REGION Network 1
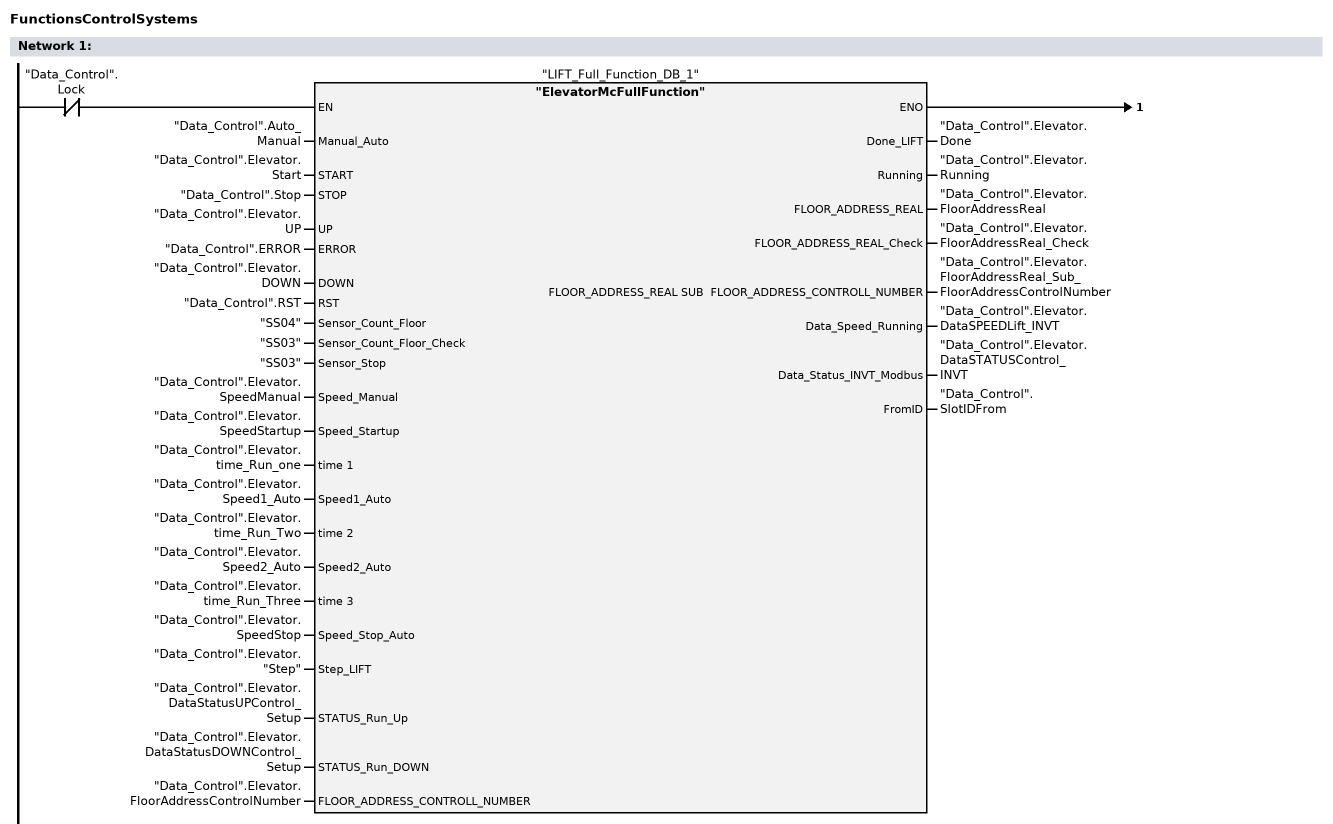
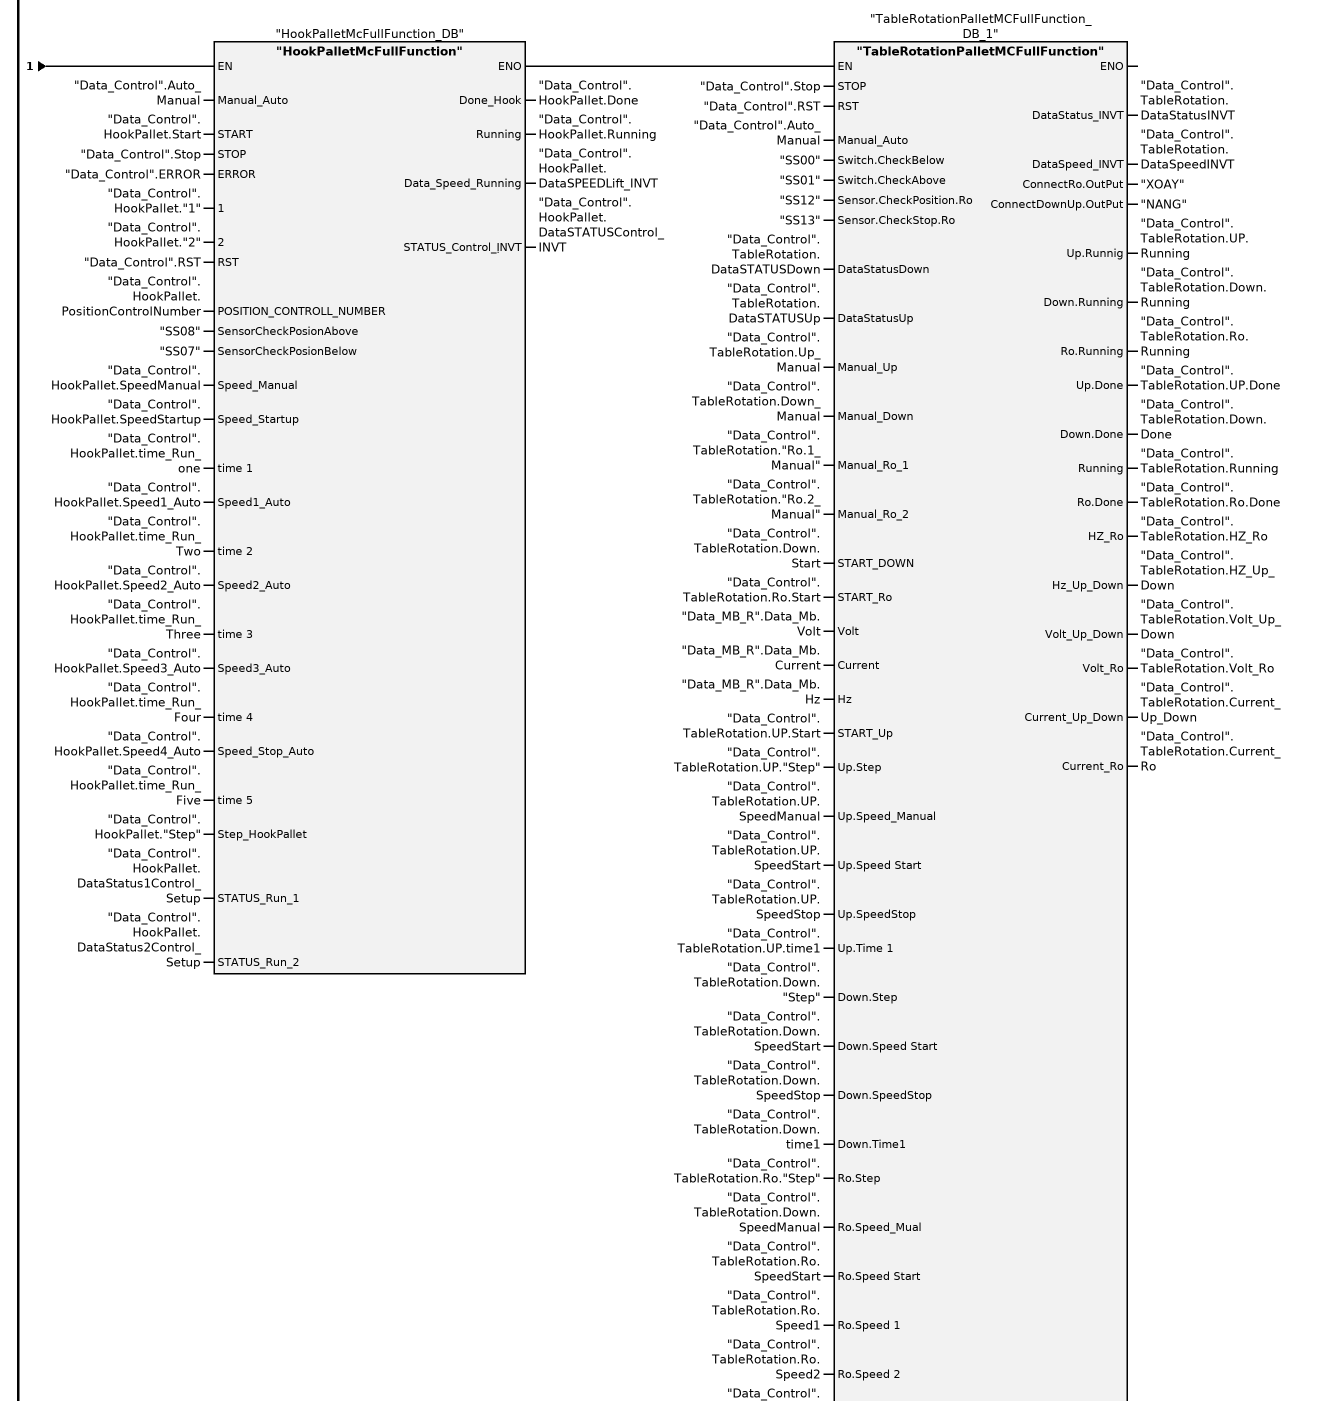
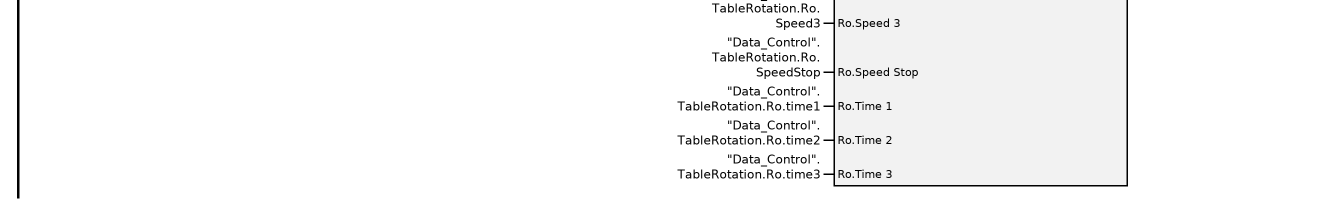
   RUNG wire#powerrail
      I_Contact( "Data_Control".Lock )
      "LIFT_Full_Function_DB_1"(Manual_Auto := "Data_Control".Auto_Manual, START := "Data_Control".Elevator.Start, STOP := "Data_Control".Stop, UP := "Data_Control".Elevator.UP, ERROR := "Data_Control".ERROR, DOWN := "Data_Control".Elevator.DOWN, RST := "Data_Control".RST, Sensor_Count_Floor := "SS04", Sensor_Count_Floor_Check := "SS03", Sensor_Stop := "SS03", Speed_Manual := "Data_Control".Elevator.SpeedManual, Speed_Startup := "Data_Control".Elevator.SpeedStartup, "time 1" := "Data_Control".Elevator.time_Run_one, Speed1_Auto := "Data_Control".Elevator.Speed1_Auto, "time 2" := "Data_Control".Elevator.time_Run_Two, Speed2_Auto := "Data_Control".Elevator.Speed2_Auto, "time 3" := "Data_Control".Elevator.time_Run_Three, Speed_Stop_Auto := "Data_Control".Elevator.SpeedStop, Step_LIFT := "Data_Control".Elevator."Step", STATUS_Run_Up := "Data_Control".Elevator.DataStatusUPControl_Setup, STATUS_Run_DOWN := "Data_Control".Elevator.DataStatusDOWNControl_Setup, FLOOR_ADDRESS_CONTROLL_NUMBER := "Data_Control".Elevator.FloorAddressControlNumber, Done_LIFT => "Data_Control".Elevator.Done, Running => "Data_Control".Elevator.Running, FLOOR_ADDRESS_REAL => "Data_Control".Elevator.FloorAddressReal, FLOOR_ADDRESS_REAL_Check => "Data_Control".Elevator.FloorAddressReal_Check, "FLOOR_ADDRESS_REAL SUB  FLOOR_ADDRESS_CONTROLL_NUMBER" => "Data_Control".Elevator.FloorAddressReal_Sub_FloorAddressControlNumber, Data_Speed_Running => "Data_Control".Elevator.DataSPEEDLift_INVT, Data_Status_INVT_Modbus => "Data_Control".Elevator.DataSTATUSControl_INVT, FromID => "Data_Control".SlotIDFrom)
      "HookPalletMcFullFunction_DB"(Manual_Auto := "Data_Control".Auto_Manual, START := "Data_Control".HookPallet.Start, STOP := "Data_Control".Stop, ERROR := "Data_Control".ERROR, "1" := "Data_Control".HookPallet."1", "2" := "Data_Control".HookPallet."2", RST := "Data_Control".RST, POSITION_CONTROLL_NUMBER := "Data_Control".HookPallet.PositionControlNumber, SensorCheckPosionAbove := "SS08", SensorCheckPosionBelow := "SS07", Speed_Manual := "Data_Control".HookPallet.SpeedManual, Speed_Startup := "Data_Control".HookPallet.SpeedStartup, "time 1" := "Data_Control".HookPallet.time_Run_one, Speed1_Auto := "Data_Control".HookPallet.Speed1_Auto, "time 2" := "Data_Control".HookPallet.time_Run_Two, Speed2_Auto := "Data_Control".HookPallet.Speed2_Auto, "time 3" := "Data_Control".HookPallet.time_Run_Three, Speed3_Auto := "Data_Control".HookPallet.Speed3_Auto, "time 4" := "Data_Control".HookPallet.time_Run_Four, Speed_Stop_Auto := "Data_Control".HookPallet.Speed4_Auto, "time 5" := "Data_Control".HookPallet.time_Run_Five, Step_HookPallet := "Data_Control".HookPallet."Step", STATUS_Run_1 := "Data_Control".HookPallet.DataStatus1Control_Setup, STATUS_Run_2 := "Data_Control".HookPallet.DataStatus2Control_Setup, Done_Hook => "Data_Control".HookPallet.Done, Running => "Data_Control".HookPallet.Running, Data_Speed_Running => "Data_Control".HookPallet.DataSPEEDLift_INVT, STATUS_Control_ỊNVT => "Data_Control".HookPallet.DataSTATUSControl_INVT)
      "TableRotationPalletMCFullFunction_DB_1"(STOP := "Data_Control".Stop, RST := "Data_Control".RST, Manual_Auto := "Data_Control".Auto_Manual, "Switch.CheckBelow" := "SS00", "Switch.CheckAbove" := "SS01", "Sensor.CheckPosition.Ro" := "SS12", "Sensor.CheckStop.Ro" := "SS13", DataStatusDown := "Data_Control".TableRotation.DataSTATUSDown, DataStatusUp := "Data_Control".TableRotation.DataSTATUSUp, Manual_Up := "Data_Control".TableRotation.Up_Manual, Manual_Down := "Data_Control".TableRotation.Down_Manual, Manual_Ro_1 := "Data_Control".TableRotation."Ro.1_Manual", Manual_Ro_2 := "Data_Control".TableRotation."Ro.2_Manual", START_DOWN := "Data_Control".TableRotation.Down.Start, START_Ro := "Data_Control".TableRotation.Ro.Start, Volt := "Data_MB_R".Data_Mb.Volt, Current := "Data_MB_R".Data_Mb.Current, Hz := "Data_MB_R".Data_Mb.Hz, START_Up := "Data_Control".TableRotation.UP.Start, "Up.Step" := "Data_Control".TableRotation.UP."Step", "Up.Speed_Manual" := "Data_Control".TableRotation.UP.SpeedManual, "Up.Speed Start" := "Data_Control".TableRotation.UP.SpeedStart, "Up.SpeedStop" := "Data_Control".TableRotation.UP.SpeedStop, "Up.Time 1" := "Data_Control".TableRotation.UP.time1, "Down.Step" := "Data_Control".TableRotation.Down."Step", "Down.Speed Start" := "Data_Control".TableRotation.Down.SpeedStart, "Down.SpeedStop" := "Data_Control".TableRotation.Down.SpeedStop, "Down.Time1" := "Data_Control".TableRotation.Down.time1, "Ro.Step" := "Data_Control".TableRotation.Ro."Step", "Ro.Speed_Mual" := "Data_Control".TableRotation.Down.SpeedManual, "Ro.Speed Start" := "Data_Control".TableRotation.Ro.SpeedStart, "Ro.Speed 1" := "Data_Control".TableRotation.Ro.Speed1, "Ro.Speed 2" := "Data_Control".TableRotation.Ro.Speed2, "Ro.Speed 3" := "Data_Control".TableRotation.Ro.Speed3, "Ro.Speed Stop" := "Data_Control".TableRotation.Ro.SpeedStop, "Ro.Time 1" := "Data_Control".TableRotation.Ro.time1, "Ro.Time 2" := "Data_Control".TableRotation.Ro.time2, "Ro.Time 3" := "Data_Control".TableRotation.Ro.time3, DataStatus_INVT => "Data_Control".TableRotation.DataStatusINVT, DataSpeed_INVT => "Data_Control".TableRotation.DataSpeedINVT, "ConnectRo.OutPut" => "XOAY", "ConnectDownUp.OutPut" => "NANG", "Up.Runnig" => "Data_Control".TableRotation.UP.Running, "Down.Running" => "Data_Control".TableRotation.Down.Running, "Ro.Running" => "Data_Control".TableRotation.Ro.Running, "Up.Done" => "Data_Control".TableRotation.UP.Done, "Down.Done" => "Data_Control".TableRotation.Down.Done, Running => "Data_Control".TableRotation.Running, "Ro.Done" => "Data_Control".TableRotation.Ro.Done, HZ_Ro => "Data_Control".TableRotation.HZ_Ro, Hz_Up_Down => "Data_Control".TableRotation.HZ_Up_Down, Volt_Up_Down => "Data_Control".TableRotation.Volt_Up_Down, Volt_Ro => "Data_Control".TableRotation.Volt_Ro, Current_Up_Down => "Data_Control".TableRotation.Current_Up_Down, Current_Ro => "Data_Control".TableRotation.Current_Ro)
   END_RUNG
   // the same network as SCL:
   "LIFT_Full_Function_DB_1"(EN := NOT "Data_Control".Lock,   // "ElevatorMcFullFunction"
                           Manual_Auto := "Data_Control".Auto_Manual,
                           START := "Data_Control".Elevator.Start,
                           STOP := "Data_Control".Stop,
                           UP := "Data_Control".Elevator.UP,
                           ERROR := "Data_Control".ERROR,
                           DOWN := "Data_Control".Elevator.DOWN,
                           RST := "Data_Control".RST,
                           Sensor_Count_Floor := "SS04",
                           Sensor_Count_Floor_Check := "SS03",
                           Sensor_Stop := "SS03",
                           Speed_Manual := "Data_Control".Elevator.SpeedManual,
                           Speed_Startup := "Data_Control".Elevator.SpeedStartup,
                           "time 1" := "Data_Control".Elevator.time_Run_one,
                           Speed1_Auto := "Data_Control".Elevator.Speed1_Auto,
                           "time 2" := "Data_Control".Elevator.time_Run_Two,
                           Speed2_Auto := "Data_Control".Elevator.Speed2_Auto,
                           "time 3" := "Data_Control".Elevator.time_Run_Three,
                           Speed_Stop_Auto := "Data_Control".Elevator.SpeedStop,
                           Step_LIFT := "Data_Control".Elevator."Step",
                           STATUS_Run_Up := "Data_Control".Elevator.DataStatusUPControl_Setup,
                           STATUS_Run_DOWN := "Data_Control".Elevator.DataStatusDOWNControl_Setup,
                           FLOOR_ADDRESS_CONTROLL_NUMBER := "Data_Control".Elevator.FloorAddressControlNumber,
                           Done_LIFT => "Data_Control".Elevator.Done,
                           Running => "Data_Control".Elevator.Running,
                           FLOOR_ADDRESS_REAL => "Data_Control".Elevator.FloorAddressReal,
                           FLOOR_ADDRESS_REAL_Check => "Data_Control".Elevator.FloorAddressReal_Check,
                           "FLOOR_ADDRESS_REAL SUB  FLOOR_ADDRESS_CONTROLL_NUMBER" => "Data_Control".Elevator.FloorAddressReal_Sub_FloorAddressControlNumber,
                           Data_Speed_Running => "Data_Control".Elevator.DataSPEEDLift_INVT,
                           Data_Status_INVT_Modbus => "Data_Control".Elevator.DataSTATUSControl_INVT,
                           FromID => "Data_Control".SlotIDFrom,
                           ENO => #_w1);
   "HookPalletMcFullFunction_DB"(EN := #_w1,   // "HookPalletMcFullFunction"
                           Manual_Auto := "Data_Control".Auto_Manual,
                           START := "Data_Control".HookPallet.Start,
                           STOP := "Data_Control".Stop,
                           ERROR := "Data_Control".ERROR,
                           "1" := "Data_Control".HookPallet."1",
                           "2" := "Data_Control".HookPallet."2",
                           RST := "Data_Control".RST,
                           POSITION_CONTROLL_NUMBER := "Data_Control".HookPallet.PositionControlNumber,
                           SensorCheckPosionAbove := "SS08",
                           SensorCheckPosionBelow := "SS07",
                           Speed_Manual := "Data_Control".HookPallet.SpeedManual,
                           Speed_Startup := "Data_Control".HookPallet.SpeedStartup,
                           "time 1" := "Data_Control".HookPallet.time_Run_one,
                           Speed1_Auto := "Data_Control".HookPallet.Speed1_Auto,
                           "time 2" := "Data_Control".HookPallet.time_Run_Two,
                           Speed2_Auto := "Data_Control".HookPallet.Speed2_Auto,
                           "time 3" := "Data_Control".HookPallet.time_Run_Three,
                           Speed3_Auto := "Data_Control".HookPallet.Speed3_Auto,
                           "time 4" := "Data_Control".HookPallet.time_Run_Four,
                           Speed_Stop_Auto := "Data_Control".HookPallet.Speed4_Auto,
                           "time 5" := "Data_Control".HookPallet.time_Run_Five,
                           Step_HookPallet := "Data_Control".HookPallet."Step",
                           STATUS_Run_1 := "Data_Control".HookPallet.DataStatus1Control_Setup,
                           STATUS_Run_2 := "Data_Control".HookPallet.DataStatus2Control_Setup,
                           Done_Hook => "Data_Control".HookPallet.Done,
                           Running => "Data_Control".HookPallet.Running,
                           Data_Speed_Running => "Data_Control".HookPallet.DataSPEEDLift_INVT,
                           STATUS_Control_ỊNVT => "Data_Control".HookPallet.DataSTATUSControl_INVT,
                           ENO => #_w2);
   IF #_w2 THEN
       "TableRotationPalletMCFullFunction_DB_1"(STOP := "Data_Control".Stop,   // "TableRotationPalletMCFullFunction"
                               RST := "Data_Control".RST,
                               Manual_Auto := "Data_Control".Auto_Manual,
                               "Switch.CheckBelow" := "SS00",
                               "Switch.CheckAbove" := "SS01",
                               "Sensor.CheckPosition.Ro" := "SS12",
                               "Sensor.CheckStop.Ro" := "SS13",
                               DataStatusDown := "Data_Control".TableRotation.DataSTATUSDown,
                               DataStatusUp := "Data_Control".TableRotation.DataSTATUSUp,
                               Manual_Up := "Data_Control".TableRotation.Up_Manual,
                               Manual_Down := "Data_Control".TableRotation.Down_Manual,
                               Manual_Ro_1 := "Data_Control".TableRotation."Ro.1_Manual",
                               Manual_Ro_2 := "Data_Control".TableRotation."Ro.2_Manual",
                               START_DOWN := "Data_Control".TableRotation.Down.Start,
                               START_Ro := "Data_Control".TableRotation.Ro.Start,
                               Volt := "Data_MB_R".Data_Mb.Volt,
                               Current := "Data_MB_R".Data_Mb.Current,
                               Hz := "Data_MB_R".Data_Mb.Hz,
                               START_Up := "Data_Control".TableRotation.UP.Start,
                               "Up.Step" := "Data_Control".TableRotation.UP."Step",
                               "Up.Speed_Manual" := "Data_Control".TableRotation.UP.SpeedManual,
                               "Up.Speed Start" := "Data_Control".TableRotation.UP.SpeedStart,
                               "Up.SpeedStop" := "Data_Control".TableRotation.UP.SpeedStop,
                               "Up.Time 1" := "Data_Control".TableRotation.UP.time1,
                               "Down.Step" := "Data_Control".TableRotation.Down."Step",
                               "Down.Speed Start" := "Data_Control".TableRotation.Down.SpeedStart,
                               "Down.SpeedStop" := "Data_Control".TableRotation.Down.SpeedStop,
                               "Down.Time1" := "Data_Control".TableRotation.Down.time1,
                               "Ro.Step" := "Data_Control".TableRotation.Ro."Step",
                               "Ro.Speed_Mual" := "Data_Control".TableRotation.Down.SpeedManual,
                               "Ro.Speed Start" := "Data_Control".TableRotation.Ro.SpeedStart,
                               "Ro.Speed 1" := "Data_Control".TableRotation.Ro.Speed1,
                               "Ro.Speed 2" := "Data_Control".TableRotation.Ro.Speed2,
                               "Ro.Speed 3" := "Data_Control".TableRotation.Ro.Speed3,
                               "Ro.Speed Stop" := "Data_Control".TableRotation.Ro.SpeedStop,
                               "Ro.Time 1" := "Data_Control".TableRotation.Ro.time1,
                               "Ro.Time 2" := "Data_Control".TableRotation.Ro.time2,
                               "Ro.Time 3" := "Data_Control".TableRotation.Ro.time3,
                               DataStatus_INVT => "Data_Control".TableRotation.DataStatusINVT,
                               DataSpeed_INVT => "Data_Control".TableRotation.DataSpeedINVT,
                               "ConnectRo.OutPut" => "XOAY",
                               "ConnectDownUp.OutPut" => "NANG",
                               "Up.Runnig" => "Data_Control".TableRotation.UP.Running,
                               "Down.Running" => "Data_Control".TableRotation.Down.Running,
                               "Ro.Running" => "Data_Control".TableRotation.Ro.Running,
                               "Up.Done" => "Data_Control".TableRotation.UP.Done,
                               "Down.Done" => "Data_Control".TableRotation.Down.Done,
                               Running => "Data_Control".TableRotation.Running,
                               "Ro.Done" => "Data_Control".TableRotation.Ro.Done,
                               HZ_Ro => "Data_Control".TableRotation.HZ_Ro,
                               Hz_Up_Down => "Data_Control".TableRotation.HZ_Up_Down,
                               Volt_Up_Down => "Data_Control".TableRotation.Volt_Up_Down,
                               Volt_Ro => "Data_Control".TableRotation.Volt_Ro,
                               Current_Up_Down => "Data_Control".TableRotation.Current_Up_Down,
                               Current_Ro => "Data_Control".TableRotation.Current_Ro);
   END_IF;
END_REGION
END_FUNCTION_BLOCK

FUNCTION_BLOCK "HookPalletMcFullFunction"   // FB27, LAD
{ S7_Optimized_Access := 'TRUE' }
VERSION : 0.1
   VAR_INPUT
      Manual_Auto : Bool;
      START : Bool;
      STOP : Bool;
      ERROR : Bool;
      "1" : Bool;
      "2" : Bool;
      RST : Bool;
      POSITION_CONTROLL_NUMBER : Int;   // address Elevator use to control
      SensorCheckPosionAbove : Bool;   // it have a Pallet
      SensorCheckPosionBelow : Bool;   // it have not Pallet
      Speed_Manual : Int;
      Speed_Startup : Int;
      "time 1" : Time;
      Speed1_Auto : Int;
      "time 2" : Time;
      Speed2_Auto : Int;
      "time 3" : Time;
      Speed3_Auto : Int;
      "time 4" : Time;
      Speed_Stop_Auto : Int;
      "time 5" : Time;
   END_VAR
   VAR_OUTPUT
      Done_Hook : Bool;
      Running : Bool;   // Lift Running
      Data_Speed_Running : Int;
      STATUS_Control_ỊNVT : Word;
   END_VAR
   VAR_IN_OUT
      Step_HookPallet : Int;   // steps used to control
      STATUS_Run_1 : Word := 16#0002;   // Set_Up Run R/F
      STATUS_Run_2 : Word := 16#0004;   // Set_Up Run R/F
   END_VAR
   VAR_TEMP   // added for the SCL form of the ladder/FBD networks
      _w1 : Bool;
   END_VAR
BEGIN

REGION Network 1
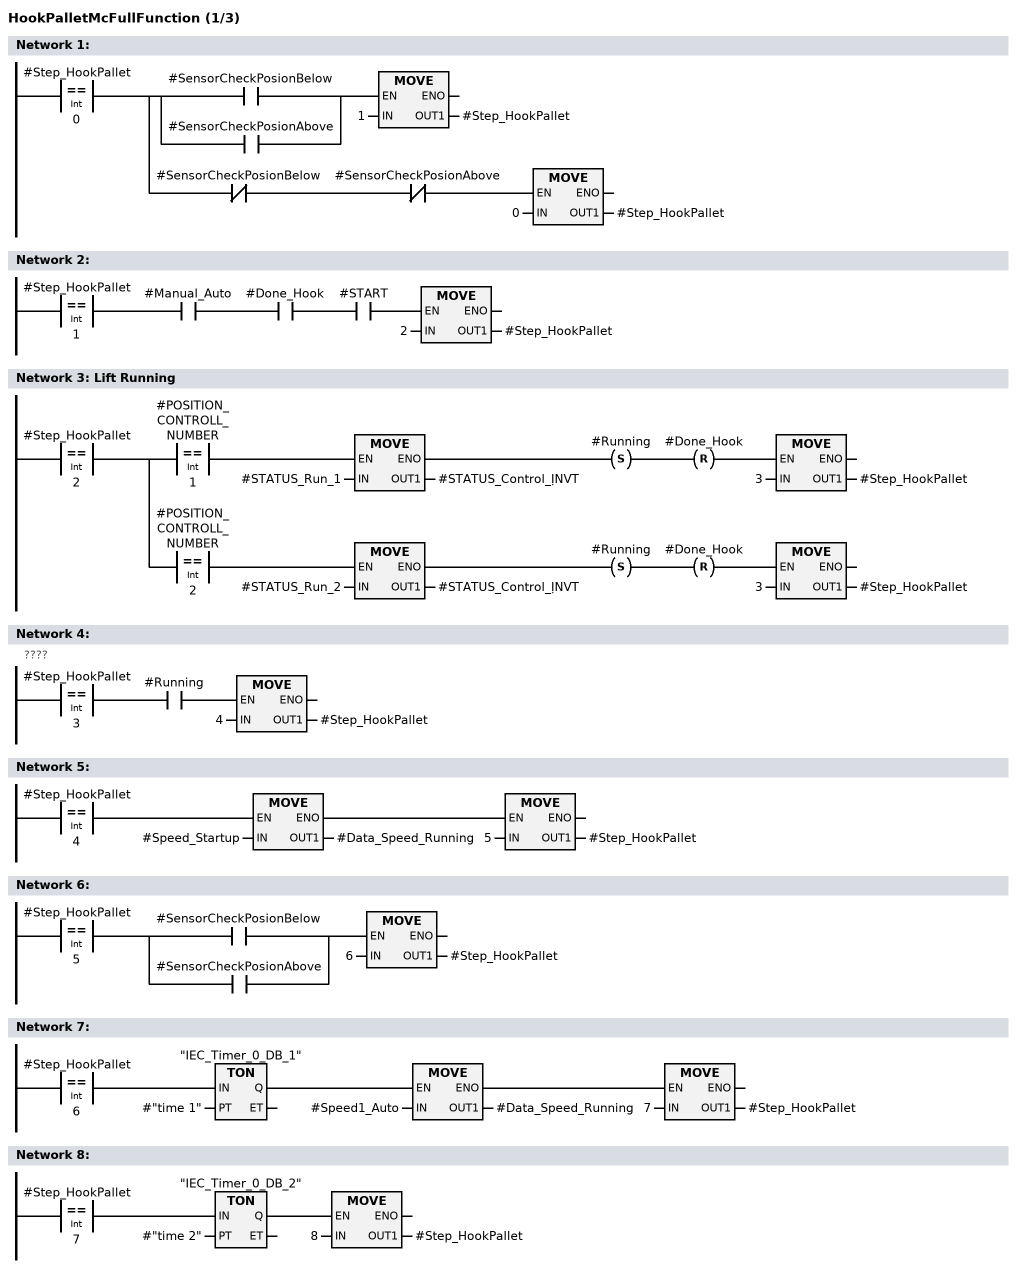
   RUNG wire#powerrail
      { S7_Templates := "SrcType := Int" } EQ_Contact(in1 := #Step_HookPallet, in2 := 0)
      wire#w1
      Contact( #SensorCheckPosionBelow )
      wire#w2
      Move(in := 1, out1 => #Step_HookPallet)
   END_RUNG
   RUNG wire#w1
      Contact( #SensorCheckPosionAbove )
   END_RUNG wire#w2
   RUNG wire#w1
      I_Contact( #SensorCheckPosionBelow )
      I_Contact( #SensorCheckPosionAbove )
      Move(in := 0, out1 => #Step_HookPallet)
   END_RUNG
   // the same network as SCL:
   #_w1 := #Step_HookPallet = 0;
   IF #_w1 AND (#SensorCheckPosionBelow OR #SensorCheckPosionAbove) THEN #Step_HookPallet := 1; END_IF;
   IF #_w1 AND NOT #SensorCheckPosionBelow AND NOT #SensorCheckPosionAbove THEN
       #Step_HookPallet := 0;
   END_IF;
END_REGION

REGION Network 2
   RUNG wire#powerrail
      { S7_Templates := "SrcType := Int" } EQ_Contact(in1 := #Step_HookPallet, in2 := 1)
      Contact( #Manual_Auto )
      Contact( #Done_Hook )
      Contact( #START )
      Move(in := 2, out1 => #Step_HookPallet)
   END_RUNG
   // the same network as SCL:
   IF (#Step_HookPallet = 1) AND #Manual_Auto AND #Done_Hook AND #START THEN #Step_HookPallet := 2; END_IF;
END_REGION

REGION Network 3: Lift Running
   RUNG wire#powerrail
      { S7_Templates := "SrcType := Int" } EQ_Contact(in1 := #Step_HookPallet, in2 := 2)
      wire#w1
      { S7_Templates := "SrcType := Int" } EQ_Contact(in1 := #POSITION_CONTROLL_NUMBER, in2 := 1)
      Move(in := #STATUS_Run_1, out1 => #STATUS_Control_ỊNVT)
      S_Coil( #Running )
      R_Coil( #Done_Hook )
      Move(in := 3, out1 => #Step_HookPallet)
   END_RUNG
   RUNG wire#w1
      { S7_Templates := "SrcType := Int" } EQ_Contact(in1 := #POSITION_CONTROLL_NUMBER, in2 := 2)
      Move(in := #STATUS_Run_2, out1 => #STATUS_Control_ỊNVT)
      S_Coil( #Running )
      R_Coil( #Done_Hook )
      Move(in := 3, out1 => #Step_HookPallet)
   END_RUNG
   // the same network as SCL:
   #_w1 := #Step_HookPallet = 2;
   IF #_w1 AND (#POSITION_CONTROLL_NUMBER = 1) THEN
       #STATUS_Control_ỊNVT := #STATUS_Run_1;
       #Running := TRUE;
       #Done_Hook := FALSE;
       #Step_HookPallet := 3;
   END_IF;
   IF #_w1 AND (#POSITION_CONTROLL_NUMBER = 2) THEN
       #STATUS_Control_ỊNVT := #STATUS_Run_2;
       #Running := TRUE;
       #Done_Hook := FALSE;
       #Step_HookPallet := 3;
   END_IF;
END_REGION

REGION Network 4
   // ????
   RUNG wire#powerrail
      { S7_Templates := "SrcType := Int" } EQ_Contact(in1 := #Step_HookPallet, in2 := 3)
      Contact( #Running )
      Move(in := 4, out1 => #Step_HookPallet)
   END_RUNG
   // the same network as SCL:
   IF (#Step_HookPallet = 3) AND #Running THEN #Step_HookPallet := 4; END_IF;
END_REGION

REGION Network 5
   RUNG wire#powerrail
      { S7_Templates := "SrcType := Int" } EQ_Contact(in1 := #Step_HookPallet, in2 := 4)
      Move(in := #Speed_Startup, out1 => #Data_Speed_Running)
      Move(in := 5, out1 => #Step_HookPallet)
   END_RUNG
   // the same network as SCL:
   IF #Step_HookPallet = 4 THEN
       #Data_Speed_Running := #Speed_Startup;
       #Step_HookPallet := 5;
   END_IF;
END_REGION

REGION Network 6
   RUNG wire#powerrail
      { S7_Templates := "SrcType := Int" } EQ_Contact(in1 := #Step_HookPallet, in2 := 5)
      wire#w1
      Contact( #SensorCheckPosionBelow )
      wire#w2
      Move(in := 6, out1 => #Step_HookPallet)
   END_RUNG
   RUNG wire#w1
      Contact( #SensorCheckPosionAbove )
   END_RUNG wire#w2
   // the same network as SCL:
   IF (#Step_HookPallet = 5) AND (#SensorCheckPosionBelow OR #SensorCheckPosionAbove) THEN
       #Step_HookPallet := 6;
   END_IF;
END_REGION

REGION Network 7
   "IEC_Timer_0_DB_1".TON(IN := #Step_HookPallet = 6, PT := #"time 1");
   IF "IEC_Timer_0_DB_1".Q THEN
       #Data_Speed_Running := #Speed1_Auto;
       #Step_HookPallet := 7;
   END_IF;
END_REGION

REGION Network 8
   "IEC_Timer_0_DB_2".TON(IN := #Step_HookPallet = 7, PT := #"time 2");
   IF "IEC_Timer_0_DB_2".Q THEN #Step_HookPallet := 8; END_IF;
END_REGION

REGION Network 9
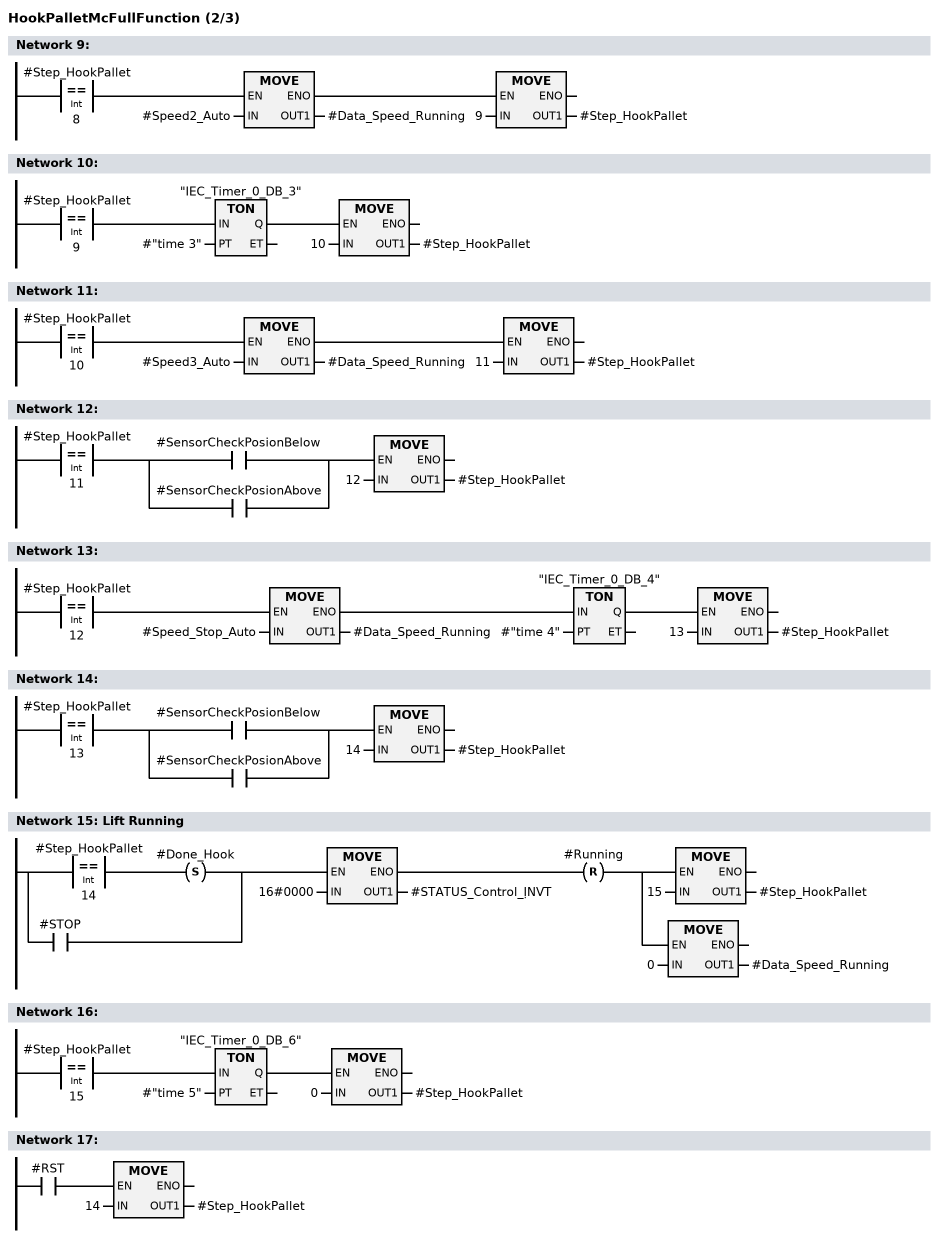
   RUNG wire#powerrail
      { S7_Templates := "SrcType := Int" } EQ_Contact(in1 := #Step_HookPallet, in2 := 8)
      Move(in := #Speed2_Auto, out1 => #Data_Speed_Running)
      Move(in := 9, out1 => #Step_HookPallet)
   END_RUNG
   // the same network as SCL:
   IF #Step_HookPallet = 8 THEN
       #Data_Speed_Running := #Speed2_Auto;
       #Step_HookPallet := 9;
   END_IF;
END_REGION

REGION Network 10
   "IEC_Timer_0_DB_3".TON(IN := #Step_HookPallet = 9, PT := #"time 3");
   IF "IEC_Timer_0_DB_3".Q THEN #Step_HookPallet := 10; END_IF;
END_REGION

REGION Network 11
   RUNG wire#powerrail
      { S7_Templates := "SrcType := Int" } EQ_Contact(in1 := #Step_HookPallet, in2 := 10)
      Move(in := #Speed3_Auto, out1 => #Data_Speed_Running)
      Move(in := 11, out1 => #Step_HookPallet)
   END_RUNG
   // the same network as SCL:
   IF #Step_HookPallet = 10 THEN
       #Data_Speed_Running := #Speed3_Auto;
       #Step_HookPallet := 11;
   END_IF;
END_REGION

REGION Network 12
   RUNG wire#powerrail
      { S7_Templates := "SrcType := Int" } EQ_Contact(in1 := #Step_HookPallet, in2 := 11)
      wire#w1
      Contact( #SensorCheckPosionBelow )
      wire#w2
      Move(in := 12, out1 => #Step_HookPallet)
   END_RUNG
   RUNG wire#w1
      Contact( #SensorCheckPosionAbove )
   END_RUNG wire#w2
   // the same network as SCL:
   IF (#Step_HookPallet = 11) AND (#SensorCheckPosionBelow OR #SensorCheckPosionAbove) THEN
       #Step_HookPallet := 12;
   END_IF;
END_REGION

REGION Network 13
   #_w1 := #Step_HookPallet = 12;
   IF #_w1 THEN #Data_Speed_Running := #Speed_Stop_Auto; END_IF;
   "IEC_Timer_0_DB_4".TON(IN := #_w1, PT := #"time 4");
   IF "IEC_Timer_0_DB_4".Q THEN #Step_HookPallet := 13; END_IF;
END_REGION

REGION Network 14
   RUNG wire#powerrail
      { S7_Templates := "SrcType := Int" } EQ_Contact(in1 := #Step_HookPallet, in2 := 13)
      wire#w1
      Contact( #SensorCheckPosionBelow )
      wire#w2
      Move(in := 14, out1 => #Step_HookPallet)
   END_RUNG
   RUNG wire#w1
      Contact( #SensorCheckPosionAbove )
   END_RUNG wire#w2
   // the same network as SCL:
   IF (#Step_HookPallet = 13) AND (#SensorCheckPosionBelow OR #SensorCheckPosionAbove) THEN
       #Step_HookPallet := 14;
   END_IF;
END_REGION

REGION Network 15: Lift Running
   RUNG wire#powerrail
      { S7_Templates := "SrcType := Int" } EQ_Contact(in1 := #Step_HookPallet, in2 := 14)
      S_Coil( #Done_Hook )
      wire#w1
      Move(in := 16#0000, out1 => #STATUS_Control_ỊNVT)
      R_Coil( #Running )
      wire#w2
      Move(in := 15, out1 => #Step_HookPallet)
   END_RUNG
   RUNG wire#powerrail
      Contact( #STOP )
   END_RUNG wire#w1
   RUNG wire#w2
      Move(in := 0, out1 => #Data_Speed_Running)
   END_RUNG
   // the same network as SCL:
   #_w1 := #Step_HookPallet = 14;
   IF #_w1 THEN #Done_Hook := TRUE; END_IF;
   IF #_w1 OR #STOP THEN
       #STATUS_Control_ỊNVT := 16#0000;
       #Running := FALSE;
       #Step_HookPallet := 15;
       #Data_Speed_Running := 0;
   END_IF;
END_REGION

REGION Network 16
   "IEC_Timer_0_DB_6".TON(IN := #Step_HookPallet = 15, PT := #"time 5");
   IF "IEC_Timer_0_DB_6".Q THEN #Step_HookPallet := 0; END_IF;
END_REGION

REGION Network 17
   RUNG wire#powerrail
      Contact( #RST )
      Move(in := 14, out1 => #Step_HookPallet)
   END_RUNG
   // the same network as SCL:
   IF #RST THEN #Step_HookPallet := 14; END_IF;
END_REGION

REGION Network 18
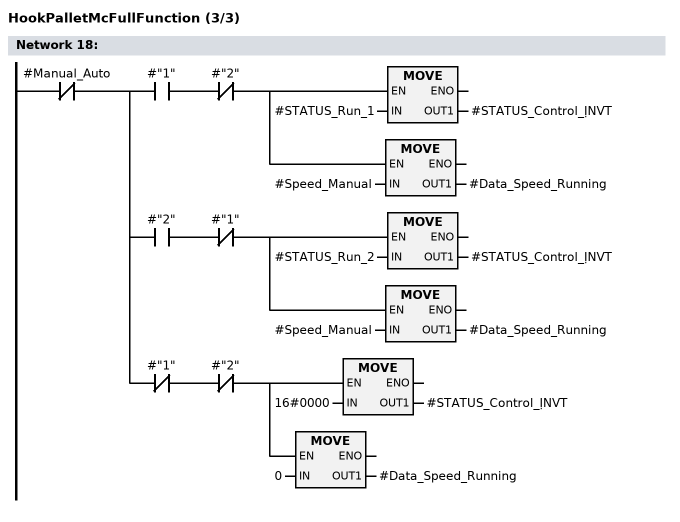
   RUNG wire#powerrail
      I_Contact( #Manual_Auto )
      wire#w1
      Contact( #"1" )
      I_Contact( #"2" )
      wire#w2
      Move(in := #STATUS_Run_1, out1 => #STATUS_Control_ỊNVT)
   END_RUNG
   RUNG wire#w2
      Move(in := #Speed_Manual, out1 => #Data_Speed_Running)
   END_RUNG
   RUNG wire#w1
      Contact( #"2" )
      I_Contact( #"1" )
      wire#w3
      Move(in := #STATUS_Run_2, out1 => #STATUS_Control_ỊNVT)
   END_RUNG
   RUNG wire#w3
      Move(in := #Speed_Manual, out1 => #Data_Speed_Running)
   END_RUNG
   RUNG wire#w1
      I_Contact( #"1" )
      I_Contact( #"2" )
      wire#w4
      Move(in := 16#0000, out1 => #STATUS_Control_ỊNVT)
   END_RUNG
   RUNG wire#w4
      Move(in := 0, out1 => #Data_Speed_Running)
   END_RUNG
   // the same network as SCL:
   IF NOT #Manual_Auto AND #"1" AND NOT #"2" THEN
       #STATUS_Control_ỊNVT := #STATUS_Run_1;
       #Data_Speed_Running := #Speed_Manual;
   END_IF;
   IF NOT #Manual_Auto AND #"2" AND NOT #"1" THEN
       #STATUS_Control_ỊNVT := #STATUS_Run_2;
       #Data_Speed_Running := #Speed_Manual;
   END_IF;
   IF NOT #Manual_Auto AND NOT #"1" AND NOT #"2" THEN
       #STATUS_Control_ỊNVT := 16#0000;
       #Data_Speed_Running := 0;
   END_IF;
END_REGION
END_FUNCTION_BLOCK

FUNCTION_BLOCK "TableRotationPalletMCFullFunction"   // FB28, LAD
{ S7_Optimized_Access := 'TRUE' }
VERSION : 0.1
   VAR_INPUT
      STOP : Bool;
      RST : Bool;
      Manual_Auto : Bool;
      "Switch.CheckBelow" : Bool;
      "Switch.CheckAbove" : Bool;
      "Sensor.CheckPosition.Ro" : Bool;
      "Sensor.CheckStop.Ro" : Bool;
      DataStatusDown : Word := 16#0002;
      DataStatusUp : Word := 16#0004;
      Manual_Up : Bool;
      Manual_Down : Bool;
      Manual_Ro_1 : Bool;
      Manual_Ro_2 : Bool;
      START_DOWN : Bool;
      START_Ro : Bool;
      Volt : Int;
      Current : Int;
      Hz : Int;
      START_Up : Bool;
   END_VAR
   VAR_OUTPUT
      DataStatus_INVT : Word;
      DataSpeed_INVT : Int;
      "ConnectRo.OutPut" : Bool;
      "ConnectDownUp.OutPut" : Bool;
      "Up.Runnig" : Bool;
      "Down.Running" : Bool;
      "Ro.Running" : Bool;
      "Up.Done" : Bool;
      "Down.Done" : Bool;
      Running : Bool;
      "Ro.Done" : Bool;
      HZ_Ro : Int;
      Hz_Up_Down : Int;
      Volt_Up_Down : Int;
      Volt_Ro : Int;
      Current_Up_Down : Int;
      Current_Ro : Int;
   END_VAR
   VAR_IN_OUT
      "Up.Step" : Int;
      "Up.Speed_Manual" : Int;
      "Up.Speed Start" : Int;
      "Up.SpeedStop" : Int;
      "Up.Time 1" : Time;
      "Down.Step" : Int;
      "Down.Speed Start" : Int;
      "Down.SpeedStop" : Int;
      "Down.Time1" : Time;
      "Ro.Step" : Int;
      "Ro.Speed_Mual" : Int;
      "Ro.Speed Start" : Int;
      "Ro.Speed 1" : Int;
      "Ro.Speed 2" : Int;
      "Ro.Speed 3" : Int;
      "Ro.Speed Stop" : Int;
      "Ro.Time 1" : Time;
      "Ro.Time 2" : Time;
      "Ro.Time 3" : Time;
   END_VAR
   VAR_TEMP   // added for the SCL form of the ladder/FBD networks
      _w1 : Bool;
      _w2 : Bool;
   END_VAR
BEGIN

REGION Network 1
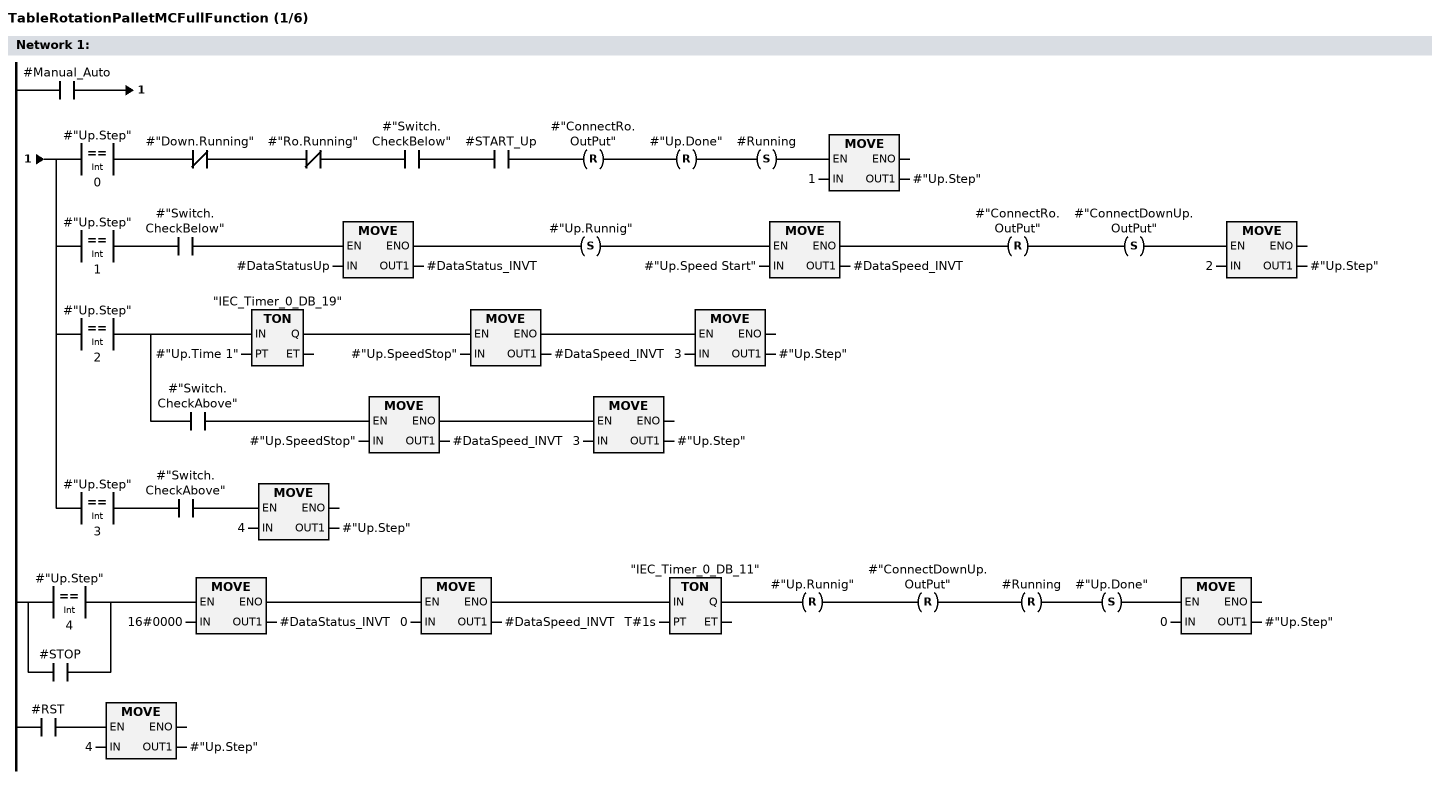
   IF #Manual_Auto AND (#"Up.Step" = 0) AND NOT #"Down.Running" AND NOT #"Ro.Running" AND #"Switch.CheckBelow" AND #START_Up THEN
       #"ConnectRo.OutPut" := FALSE;
       #"Up.Done" := FALSE;
       #Running := TRUE;
       #"Up.Step" := 1;
   END_IF;
   IF #Manual_Auto AND (#"Up.Step" = 1) AND #"Switch.CheckBelow" THEN
       #DataStatus_INVT := #DataStatusUp;
       #"Up.Runnig" := TRUE;
       #DataSpeed_INVT := #"Up.Speed Start";
       #"ConnectRo.OutPut" := FALSE;
       #"ConnectDownUp.OutPut" := TRUE;
       #"Up.Step" := 2;
   END_IF;
   #_w1 := #Manual_Auto AND (#"Up.Step" = 2);
   "IEC_Timer_0_DB_19".TON(IN := #_w1, PT := #"Up.Time 1");
   IF "IEC_Timer_0_DB_19".Q THEN
       #DataSpeed_INVT := #"Up.SpeedStop";
       #"Up.Step" := 3;
   END_IF;
   IF #_w1 AND #"Switch.CheckAbove" THEN
       #DataSpeed_INVT := #"Up.SpeedStop";
       #"Up.Step" := 3;
   END_IF;
   IF #Manual_Auto AND (#"Up.Step" = 3) AND #"Switch.CheckAbove" THEN #"Up.Step" := 4; END_IF;
   #_w2 := (#"Up.Step" = 4) OR #STOP;
   IF #_w2 THEN
       #DataStatus_INVT := 16#0000;
       #DataSpeed_INVT := 0;
   END_IF;
   "IEC_Timer_0_DB_11".TON(IN := #_w2, PT := T#1s);
   IF "IEC_Timer_0_DB_11".Q THEN
       #"Up.Runnig" := FALSE;
       #"ConnectDownUp.OutPut" := FALSE;
       #Running := FALSE;
       #"Up.Done" := TRUE;
       #"Up.Step" := 0;
   END_IF;
   IF #RST THEN #"Up.Step" := 4; END_IF;
END_REGION

REGION Network 2
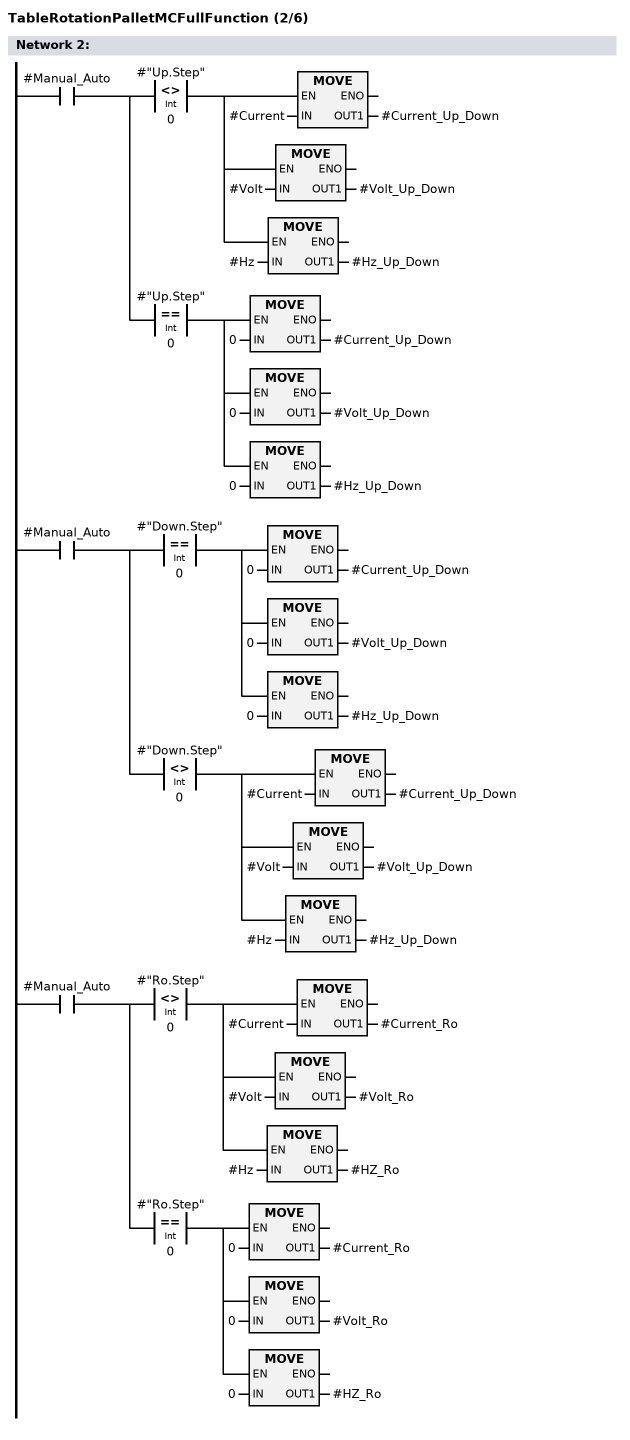
   RUNG wire#powerrail
      Contact( #Manual_Auto )
      wire#w1
      { S7_Templates := "SrcType := Int" } NE_Contact(in1 := #"Up.Step", in2 := 0)
      wire#w2
      Move(in := #Current, out1 => #Current_Up_Down)
   END_RUNG
   RUNG wire#w2
      Move(in := #Volt, out1 => #Volt_Up_Down)
   END_RUNG
   RUNG wire#w2
      Move(in := #Hz, out1 => #Hz_Up_Down)
   END_RUNG
   RUNG wire#w1
      { S7_Templates := "SrcType := Int" } EQ_Contact(in1 := #"Up.Step", in2 := 0)
      wire#w3
      Move(in := 0, out1 => #Current_Up_Down)
   END_RUNG
   RUNG wire#w3
      Move(in := 0, out1 => #Volt_Up_Down)
   END_RUNG
   RUNG wire#w3
      Move(in := 0, out1 => #Hz_Up_Down)
   END_RUNG
   RUNG wire#powerrail
      Contact( #Manual_Auto )
      wire#w4
      { S7_Templates := "SrcType := Int" } EQ_Contact(in1 := #"Down.Step", in2 := 0)
      wire#w5
      Move(in := 0, out1 => #Current_Up_Down)
   END_RUNG
   RUNG wire#w5
      Move(in := 0, out1 => #Volt_Up_Down)
   END_RUNG
   RUNG wire#w5
      Move(in := 0, out1 => #Hz_Up_Down)
   END_RUNG
   RUNG wire#w4
      { S7_Templates := "SrcType := Int" } NE_Contact(in1 := #"Down.Step", in2 := 0)
      wire#w6
      Move(in := #Current, out1 => #Current_Up_Down)
   END_RUNG
   RUNG wire#w6
      Move(in := #Volt, out1 => #Volt_Up_Down)
   END_RUNG
   RUNG wire#w6
      Move(in := #Hz, out1 => #Hz_Up_Down)
   END_RUNG
   RUNG wire#powerrail
      Contact( #Manual_Auto )
      wire#w7
      { S7_Templates := "SrcType := Int" } NE_Contact(in1 := #"Ro.Step", in2 := 0)
      wire#w8
      Move(in := #Current, out1 => #Current_Ro)
   END_RUNG
   RUNG wire#w8
      Move(in := #Volt, out1 => #Volt_Ro)
   END_RUNG
   RUNG wire#w8
      Move(in := #Hz, out1 => #HZ_Ro)
   END_RUNG
   RUNG wire#w7
      { S7_Templates := "SrcType := Int" } EQ_Contact(in1 := #"Ro.Step", in2 := 0)
      wire#w9
      Move(in := 0, out1 => #Current_Ro)
   END_RUNG
   RUNG wire#w9
      Move(in := 0, out1 => #Volt_Ro)
   END_RUNG
   RUNG wire#w9
      Move(in := 0, out1 => #HZ_Ro)
   END_RUNG
   // the same network as SCL:
   IF #Manual_Auto AND (#"Up.Step" <> 0) THEN
       #Current_Up_Down := #Current;
       #Volt_Up_Down := #Volt;
       #Hz_Up_Down := #Hz;
   END_IF;
   IF #Manual_Auto AND (#"Up.Step" = 0) THEN
       #Current_Up_Down := 0;
       #Volt_Up_Down := 0;
       #Hz_Up_Down := 0;
   END_IF;
   IF #Manual_Auto AND (#"Down.Step" = 0) THEN
       #Current_Up_Down := 0;
       #Volt_Up_Down := 0;
       #Hz_Up_Down := 0;
   END_IF;
   IF #Manual_Auto AND (#"Down.Step" <> 0) THEN
       #Current_Up_Down := #Current;
       #Volt_Up_Down := #Volt;
       #Hz_Up_Down := #Hz;
   END_IF;
   IF #Manual_Auto AND (#"Ro.Step" <> 0) THEN
       #Current_Ro := #Current;
       #Volt_Ro := #Volt;
       #HZ_Ro := #Hz;
   END_IF;
   IF #Manual_Auto AND (#"Ro.Step" = 0) THEN
       #Current_Ro := 0;
       #Volt_Ro := 0;
       #HZ_Ro := 0;
   END_IF;
END_REGION

REGION Network 3
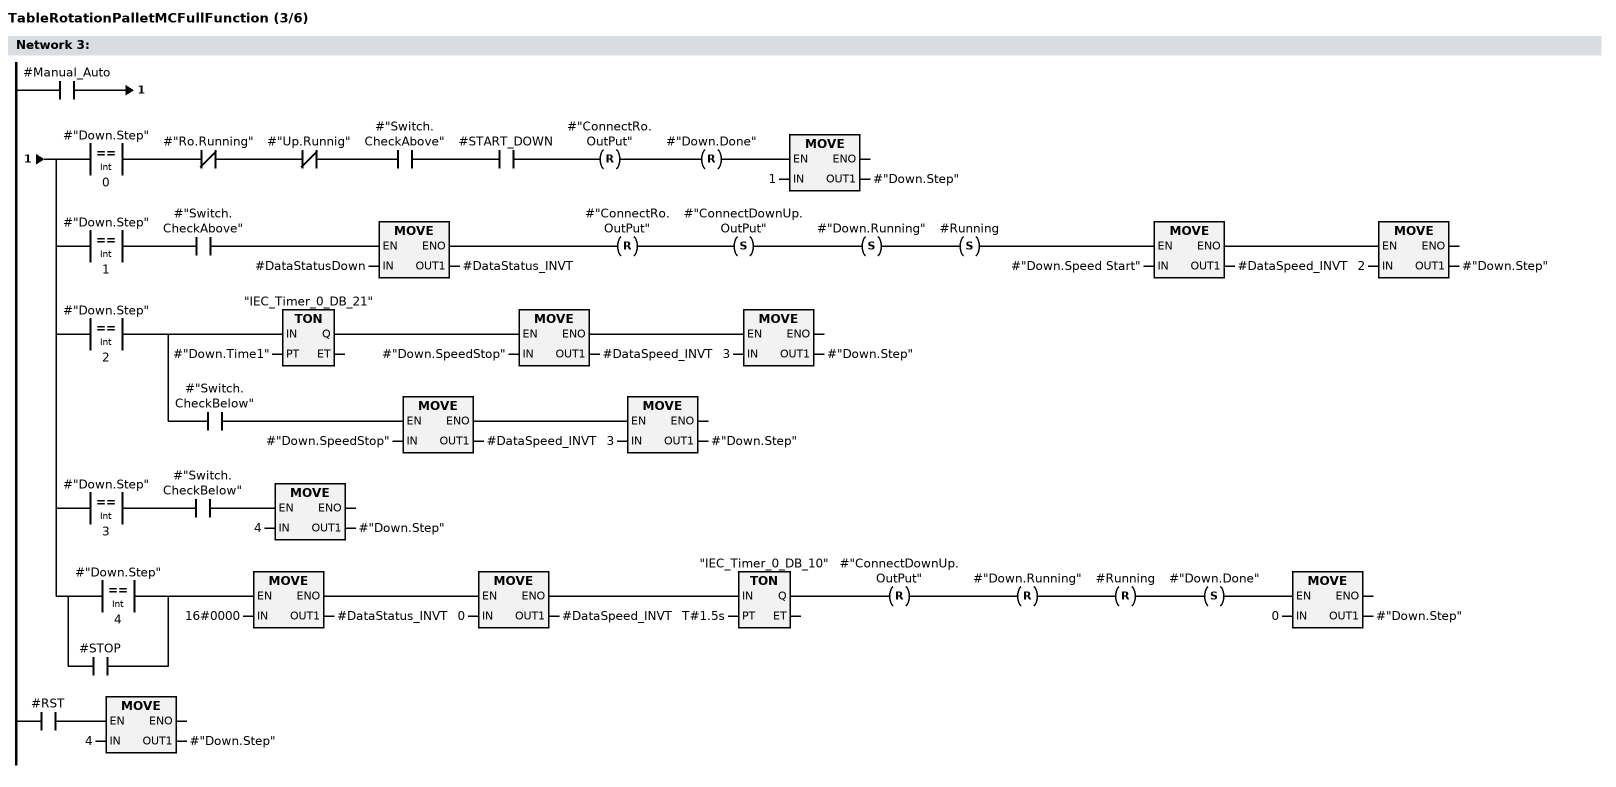
   IF #Manual_Auto AND (#"Down.Step" = 0) AND NOT #"Ro.Running" AND NOT #"Up.Runnig" AND #"Switch.CheckAbove" AND #START_DOWN THEN
       #"ConnectRo.OutPut" := FALSE;
       #"Down.Done" := FALSE;
       #"Down.Step" := 1;
   END_IF;
   IF #Manual_Auto AND (#"Down.Step" = 1) AND #"Switch.CheckAbove" THEN
       #DataStatus_INVT := #DataStatusDown;
       #"ConnectRo.OutPut" := FALSE;
       #"ConnectDownUp.OutPut" := TRUE;
       #"Down.Running" := TRUE;
       #Running := TRUE;
       #DataSpeed_INVT := #"Down.Speed Start";
       #"Down.Step" := 2;
   END_IF;
   #_w1 := #Manual_Auto AND (#"Down.Step" = 2);
   "IEC_Timer_0_DB_21".TON(IN := #_w1, PT := #"Down.Time1");
   IF "IEC_Timer_0_DB_21".Q THEN
       #DataSpeed_INVT := #"Down.SpeedStop";
       #"Down.Step" := 3;
   END_IF;
   IF #_w1 AND #"Switch.CheckBelow" THEN
       #DataSpeed_INVT := #"Down.SpeedStop";
       #"Down.Step" := 3;
   END_IF;
   IF #Manual_Auto AND (#"Down.Step" = 3) AND #"Switch.CheckBelow" THEN #"Down.Step" := 4; END_IF;
   #_w2 := #Manual_Auto AND ((#"Down.Step" = 4) OR #STOP);
   IF #_w2 THEN
       #DataStatus_INVT := 16#0000;
       #DataSpeed_INVT := 0;
   END_IF;
   "IEC_Timer_0_DB_10".TON(IN := #_w2, PT := T#1.5s);
   IF "IEC_Timer_0_DB_10".Q THEN
       #"ConnectDownUp.OutPut" := FALSE;
       #"Down.Running" := FALSE;
       #Running := FALSE;
       #"Down.Done" := TRUE;
       #"Down.Step" := 0;
   END_IF;
   IF #RST THEN #"Down.Step" := 4; END_IF;
END_REGION

REGION Network 5
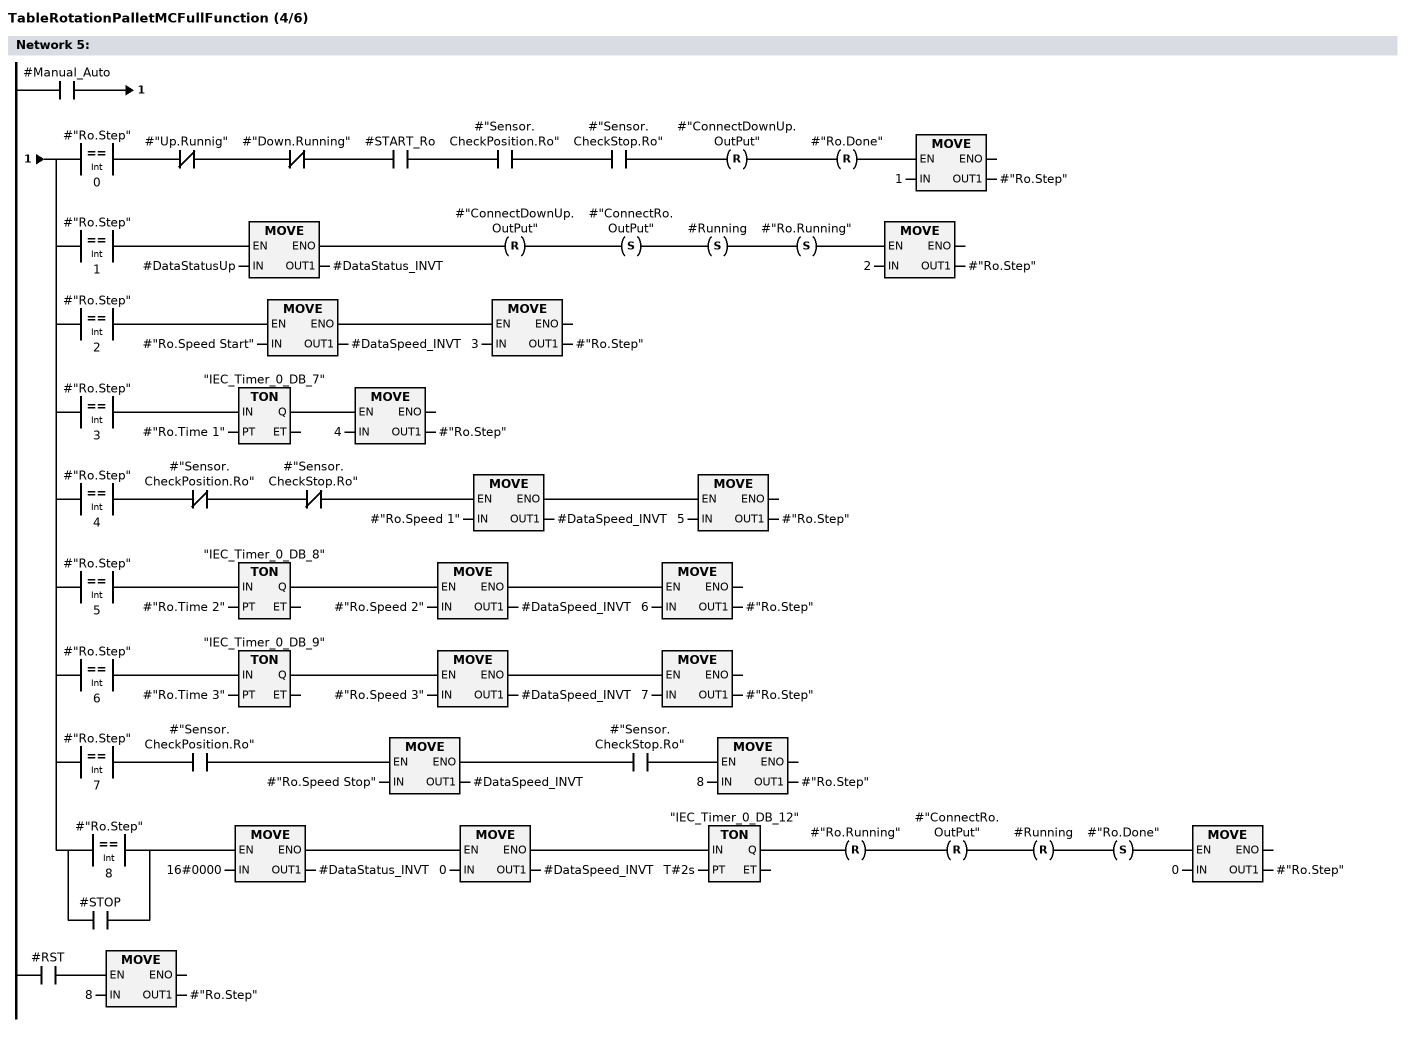
   IF #Manual_Auto AND (#"Ro.Step" = 0) AND NOT #"Up.Runnig" AND NOT #"Down.Running" AND #START_Ro AND #"Sensor.CheckPosition.Ro" AND #"Sensor.CheckStop.Ro" THEN
       #"ConnectDownUp.OutPut" := FALSE;
       #"Ro.Done" := FALSE;
       #"Ro.Step" := 1;
   END_IF;
   IF #Manual_Auto AND (#"Ro.Step" = 1) THEN
       #DataStatus_INVT := #DataStatusUp;
       #"ConnectDownUp.OutPut" := FALSE;
       #"ConnectRo.OutPut" := TRUE;
       #Running := TRUE;
       #"Ro.Running" := TRUE;
       #"Ro.Step" := 2;
   END_IF;
   IF #Manual_Auto AND (#"Ro.Step" = 2) THEN
       #DataSpeed_INVT := #"Ro.Speed Start";
       #"Ro.Step" := 3;
   END_IF;
   "IEC_Timer_0_DB_7".TON(IN := #Manual_Auto AND (#"Ro.Step" = 3), PT := #"Ro.Time 1");
   IF "IEC_Timer_0_DB_7".Q THEN #"Ro.Step" := 4; END_IF;
   IF #Manual_Auto AND (#"Ro.Step" = 4) AND NOT #"Sensor.CheckPosition.Ro" AND NOT #"Sensor.CheckStop.Ro" THEN
       #DataSpeed_INVT := #"Ro.Speed 1";
       #"Ro.Step" := 5;
   END_IF;
   "IEC_Timer_0_DB_8".TON(IN := #Manual_Auto AND (#"Ro.Step" = 5), PT := #"Ro.Time 2");
   IF "IEC_Timer_0_DB_8".Q THEN
       #DataSpeed_INVT := #"Ro.Speed 2";
       #"Ro.Step" := 6;
   END_IF;
   "IEC_Timer_0_DB_9".TON(IN := #Manual_Auto AND (#"Ro.Step" = 6), PT := #"Ro.Time 3");
   IF "IEC_Timer_0_DB_9".Q THEN
       #DataSpeed_INVT := #"Ro.Speed 3";
       #"Ro.Step" := 7;
   END_IF;
   #_w1 := #Manual_Auto AND (#"Ro.Step" = 7) AND #"Sensor.CheckPosition.Ro";
   IF #_w1 THEN #DataSpeed_INVT := #"Ro.Speed Stop"; END_IF;
   IF #_w1 AND #"Sensor.CheckStop.Ro" THEN #"Ro.Step" := 8; END_IF;
   #_w2 := #Manual_Auto AND ((#"Ro.Step" = 8) OR #STOP);
   IF #_w2 THEN
       #DataStatus_INVT := 16#0000;
       #DataSpeed_INVT := 0;
   END_IF;
   "IEC_Timer_0_DB_12".TON(IN := #_w2, PT := T#2s);
   IF "IEC_Timer_0_DB_12".Q THEN
       #"Ro.Running" := FALSE;
       #"ConnectRo.OutPut" := FALSE;
       #Running := FALSE;
       #"Ro.Done" := TRUE;
       #"Ro.Step" := 0;
   END_IF;
   IF #RST THEN #"Ro.Step" := 8; END_IF;
END_REGION

REGION Network 8
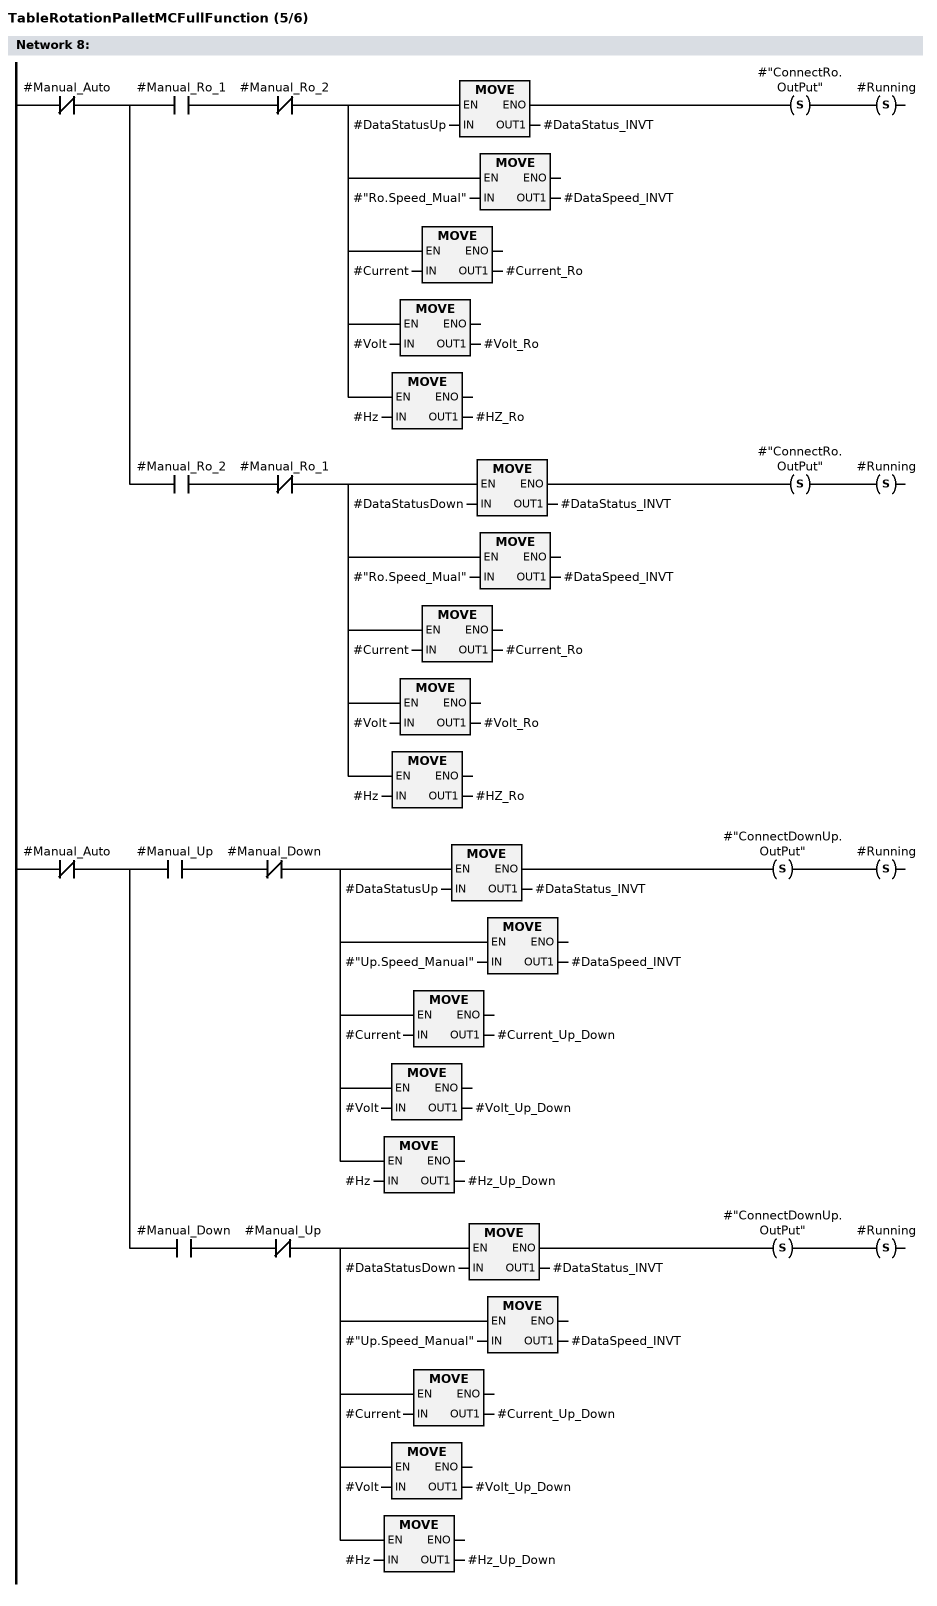
   RUNG wire#powerrail
      I_Contact( #Manual_Auto )
      wire#w1
      Contact( #Manual_Ro_1 )
      I_Contact( #Manual_Ro_2 )
      wire#w2
      Move(in := #DataStatusUp, out1 => #DataStatus_INVT)
      S_Coil( #"ConnectRo.OutPut" )
      S_Coil( #Running )
   END_RUNG
   RUNG wire#w2
      Move(in := #"Ro.Speed_Mual", out1 => #DataSpeed_INVT)
   END_RUNG
   RUNG wire#w2
      Move(in := #Current, out1 => #Current_Ro)
   END_RUNG
   RUNG wire#w2
      Move(in := #Volt, out1 => #Volt_Ro)
   END_RUNG
   RUNG wire#w2
      Move(in := #Hz, out1 => #HZ_Ro)
   END_RUNG
   RUNG wire#w1
      Contact( #Manual_Ro_2 )
      I_Contact( #Manual_Ro_1 )
      wire#w3
      Move(in := #DataStatusDown, out1 => #DataStatus_INVT)
      S_Coil( #"ConnectRo.OutPut" )
      S_Coil( #Running )
   END_RUNG
   RUNG wire#w3
      Move(in := #"Ro.Speed_Mual", out1 => #DataSpeed_INVT)
   END_RUNG
   RUNG wire#w3
      Move(in := #Current, out1 => #Current_Ro)
   END_RUNG
   RUNG wire#w3
      Move(in := #Volt, out1 => #Volt_Ro)
   END_RUNG
   RUNG wire#w3
      Move(in := #Hz, out1 => #HZ_Ro)
   END_RUNG
   RUNG wire#powerrail
      I_Contact( #Manual_Auto )
      wire#w4
      Contact( #Manual_Up )
      I_Contact( #Manual_Down )
      wire#w5
      Move(in := #DataStatusUp, out1 => #DataStatus_INVT)
      S_Coil( #"ConnectDownUp.OutPut" )
      S_Coil( #Running )
   END_RUNG
   RUNG wire#w5
      Move(in := #"Up.Speed_Manual", out1 => #DataSpeed_INVT)
   END_RUNG
   RUNG wire#w5
      Move(in := #Current, out1 => #Current_Up_Down)
   END_RUNG
   RUNG wire#w5
      Move(in := #Volt, out1 => #Volt_Up_Down)
   END_RUNG
   RUNG wire#w5
      Move(in := #Hz, out1 => #Hz_Up_Down)
   END_RUNG
   RUNG wire#w4
      Contact( #Manual_Down )
      I_Contact( #Manual_Up )
      wire#w6
      Move(in := #DataStatusDown, out1 => #DataStatus_INVT)
      S_Coil( #"ConnectDownUp.OutPut" )
      S_Coil( #Running )
   END_RUNG
   RUNG wire#w6
      Move(in := #"Up.Speed_Manual", out1 => #DataSpeed_INVT)
   END_RUNG
   RUNG wire#w6
      Move(in := #Current, out1 => #Current_Up_Down)
   END_RUNG
   RUNG wire#w6
      Move(in := #Volt, out1 => #Volt_Up_Down)
   END_RUNG
   RUNG wire#w6
      Move(in := #Hz, out1 => #Hz_Up_Down)
   END_RUNG
   // the same network as SCL:
   IF NOT #Manual_Auto AND #Manual_Ro_1 AND NOT #Manual_Ro_2 THEN
       #DataStatus_INVT := #DataStatusUp;
       #"ConnectRo.OutPut" := TRUE;
       #Running := TRUE;
       #DataSpeed_INVT := #"Ro.Speed_Mual";
       #Current_Ro := #Current;
       #Volt_Ro := #Volt;
       #HZ_Ro := #Hz;
   END_IF;
   IF NOT #Manual_Auto AND #Manual_Ro_2 AND NOT #Manual_Ro_1 THEN
       #DataStatus_INVT := #DataStatusDown;
       #"ConnectRo.OutPut" := TRUE;
       #Running := TRUE;
       #DataSpeed_INVT := #"Ro.Speed_Mual";
       #Current_Ro := #Current;
       #Volt_Ro := #Volt;
       #HZ_Ro := #Hz;
   END_IF;
   IF NOT #Manual_Auto AND #Manual_Up AND NOT #Manual_Down THEN
       #DataStatus_INVT := #DataStatusUp;
       #"ConnectDownUp.OutPut" := TRUE;
       #Running := TRUE;
       #DataSpeed_INVT := #"Up.Speed_Manual";
       #Current_Up_Down := #Current;
       #Volt_Up_Down := #Volt;
       #Hz_Up_Down := #Hz;
   END_IF;
   IF NOT #Manual_Auto AND #Manual_Down AND NOT #Manual_Up THEN
       #DataStatus_INVT := #DataStatusDown;
       #"ConnectDownUp.OutPut" := TRUE;
       #Running := TRUE;
       #DataSpeed_INVT := #"Up.Speed_Manual";
       #Current_Up_Down := #Current;
       #Volt_Up_Down := #Volt;
       #Hz_Up_Down := #Hz;
   END_IF;
END_REGION

REGION Network 9
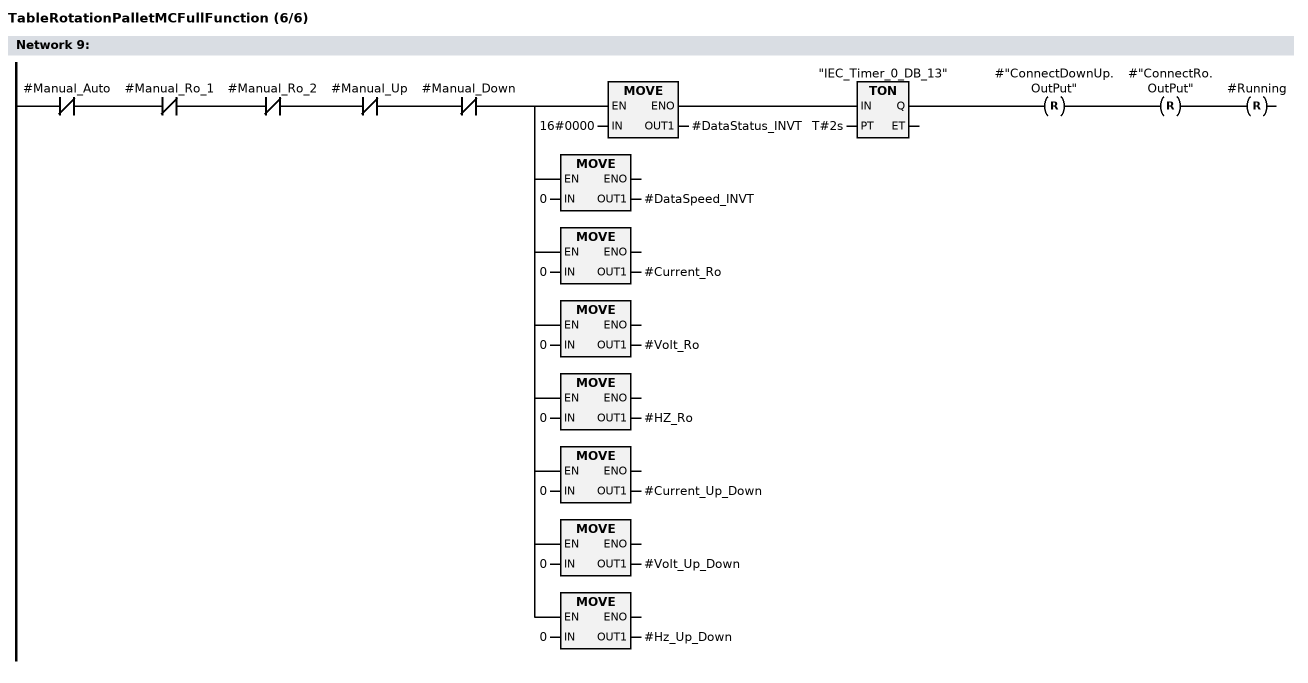
   #_w1 := NOT #Manual_Auto AND NOT #Manual_Ro_1 AND NOT #Manual_Ro_2 AND NOT #Manual_Up AND NOT #Manual_Down;
   IF #_w1 THEN #DataStatus_INVT := 16#0000; END_IF;
   "IEC_Timer_0_DB_13".TON(IN := #_w1, PT := T#2s);
   IF "IEC_Timer_0_DB_13".Q THEN
       #"ConnectDownUp.OutPut" := FALSE;
       #"ConnectRo.OutPut" := FALSE;
       #Running := FALSE;
   END_IF;
   IF #_w1 THEN
       #DataSpeed_INVT := 0;
       #Current_Ro := 0;
       #Volt_Ro := 0;
       #HZ_Ro := 0;
       #Current_Up_Down := 0;
       #Volt_Up_Down := 0;
       #Hz_Up_Down := 0;
   END_IF;
END_REGION
END_FUNCTION_BLOCK

// folder: Control/Modbus RTU

FUNCTION_BLOCK "ModbusRtu"   // FB25, LAD
{ S7_Optimized_Access := 'TRUE' }
VERSION : 0.1
BEGIN

REGION Network 1
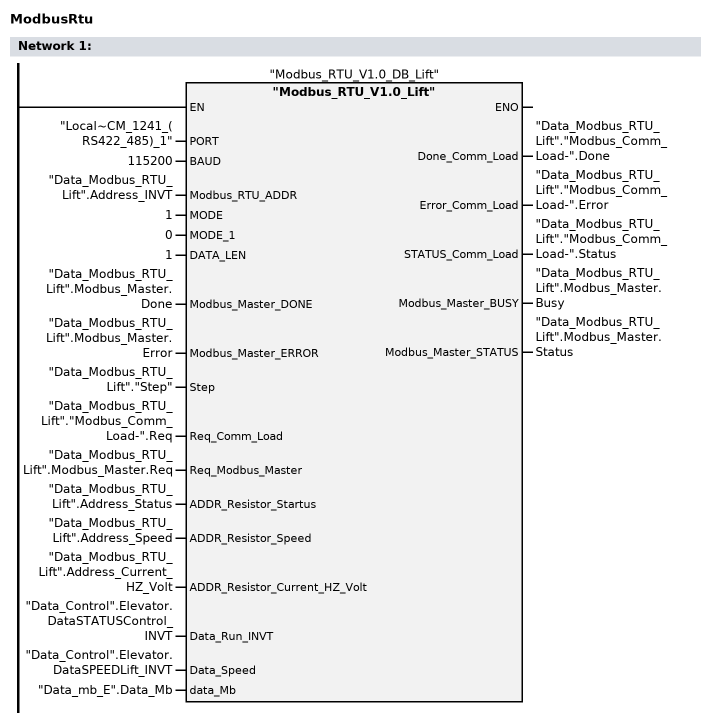
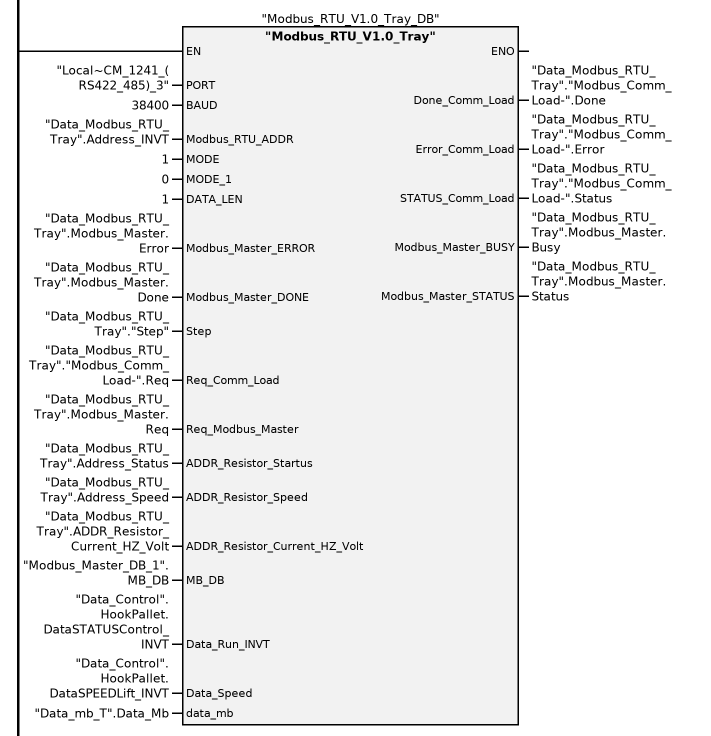
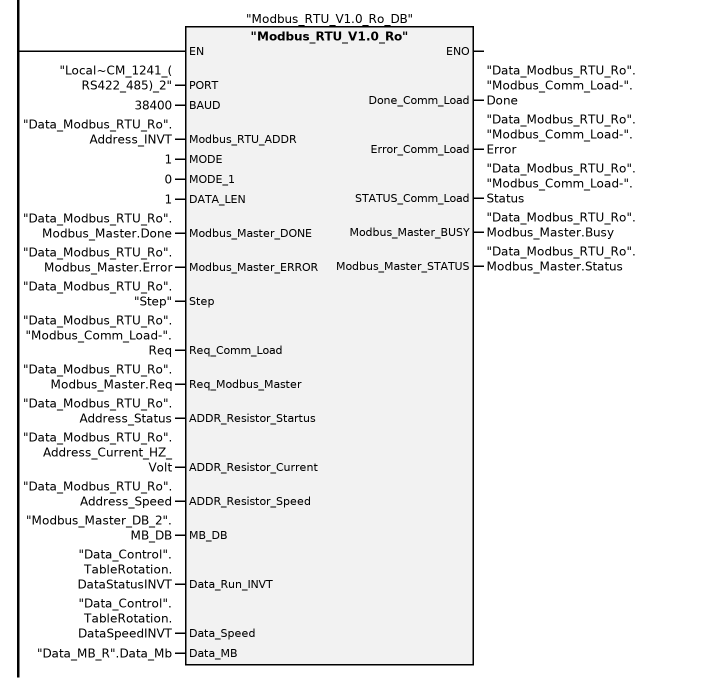
   RUNG wire#powerrail
      "Modbus_RTU_V1.0_DB_Lift"(PORT := "Local~CM_1241_(RS422_485)_1", BAUD := 115200, Modbus_RTU_ADDR := "Data_Modbus_RTU_Lift".Address_INVT, MODE := 1, MODE_1 := 0, DATA_LEN := 1, Modbus_Master_DONE := "Data_Modbus_RTU_Lift".Modbus_Master.Done, Modbus_Master_ERROR := "Data_Modbus_RTU_Lift".Modbus_Master.Error, "Step" := "Data_Modbus_RTU_Lift"."Step", Req_Comm_Load := "Data_Modbus_RTU_Lift"."Modbus_Comm_Load-".Req, Req_Modbus_Master := "Data_Modbus_RTU_Lift".Modbus_Master.Req, ADDR_Resistor_Startus := "Data_Modbus_RTU_Lift".Address_Status, ADDR_Resistor_Speed := "Data_Modbus_RTU_Lift".Address_Speed, ADDR_Resistor_Current_HZ_Volt := "Data_Modbus_RTU_Lift".Address_Current_HZ_Volt, Data_Run_INVT := "Data_Control".Elevator.DataSTATUSControl_INVT, Data_Speed := "Data_Control".Elevator.DataSPEEDLift_INVT, data_Mb := "Data_mb_E".Data_Mb, Done_Comm_Load => "Data_Modbus_RTU_Lift"."Modbus_Comm_Load-".Done, Error_Comm_Load => "Data_Modbus_RTU_Lift"."Modbus_Comm_Load-".Error, STATUS_Comm_Load => "Data_Modbus_RTU_Lift"."Modbus_Comm_Load-".Status, Modbus_Master_BUSY => "Data_Modbus_RTU_Lift".Modbus_Master.Busy, Modbus_Master_STATUS => "Data_Modbus_RTU_Lift".Modbus_Master.Status)
   END_RUNG
   RUNG wire#powerrail
      "Modbus_RTU_V1.0_Tray_DB"(PORT := "Local~CM_1241_(RS422_485)_3", BAUD := 38400, Modbus_RTU_ADDR := "Data_Modbus_RTU_Tray".Address_INVT, MODE := 1, MODE_1 := 0, DATA_LEN := 1, Modbus_Master_ERROR := "Data_Modbus_RTU_Tray".Modbus_Master.Error, Modbus_Master_DONE := "Data_Modbus_RTU_Tray".Modbus_Master.Done, "Step" := "Data_Modbus_RTU_Tray"."Step", Req_Comm_Load := "Data_Modbus_RTU_Tray"."Modbus_Comm_Load-".Req, Req_Modbus_Master := "Data_Modbus_RTU_Tray".Modbus_Master.Req, ADDR_Resistor_Startus := "Data_Modbus_RTU_Tray".Address_Status, ADDR_Resistor_Speed := "Data_Modbus_RTU_Tray".Address_Speed, ADDR_Resistor_Current_HZ_Volt := "Data_Modbus_RTU_Tray".ADDR_Resistor_Current_HZ_Volt, MB_DB := "Modbus_Master_DB_1".MB_DB, Data_Run_INVT := "Data_Control".HookPallet.DataSTATUSControl_INVT, Data_Speed := "Data_Control".HookPallet.DataSPEEDLift_INVT, data_mb := "Data_mb_T".Data_Mb, Done_Comm_Load => "Data_Modbus_RTU_Tray"."Modbus_Comm_Load-".Done, Error_Comm_Load => "Data_Modbus_RTU_Tray"."Modbus_Comm_Load-".Error, STATUS_Comm_Load => "Data_Modbus_RTU_Tray"."Modbus_Comm_Load-".Status, Modbus_Master_BUSY => "Data_Modbus_RTU_Tray".Modbus_Master.Busy, Modbus_Master_STATUS => "Data_Modbus_RTU_Tray".Modbus_Master.Status)
   END_RUNG
   RUNG wire#powerrail
      "Modbus_RTU_V1.0_Ro_DB"(PORT := "Local~CM_1241_(RS422_485)_2", BAUD := 38400, Modbus_RTU_ADDR := "Data_Modbus_RTU_Ro".Address_INVT, MODE := 1, MODE_1 := 0, DATA_LEN := 1, Modbus_Master_DONE := "Data_Modbus_RTU_Ro".Modbus_Master.Done, Modbus_Master_ERROR := "Data_Modbus_RTU_Ro".Modbus_Master.Error, "Step" := "Data_Modbus_RTU_Ro"."Step", Req_Comm_Load := "Data_Modbus_RTU_Ro"."Modbus_Comm_Load-".Req, Req_Modbus_Master := "Data_Modbus_RTU_Ro".Modbus_Master.Req, ADDR_Resistor_Startus := "Data_Modbus_RTU_Ro".Address_Status, ADDR_Resistor_Current := "Data_Modbus_RTU_Ro".Address_Current_HZ_Volt, ADDR_Resistor_Speed := "Data_Modbus_RTU_Ro".Address_Speed, MB_DB := "Modbus_Master_DB_2".MB_DB, Data_Run_INVT := "Data_Control".TableRotation.DataStatusINVT, Data_Speed := "Data_Control".TableRotation.DataSpeedINVT, Data_MB := "Data_MB_R".Data_Mb, Done_Comm_Load => "Data_Modbus_RTU_Ro"."Modbus_Comm_Load-".Done, Error_Comm_Load => "Data_Modbus_RTU_Ro"."Modbus_Comm_Load-".Error, STATUS_Comm_Load => "Data_Modbus_RTU_Ro"."Modbus_Comm_Load-".Status, Modbus_Master_BUSY => "Data_Modbus_RTU_Ro".Modbus_Master.Busy, Modbus_Master_STATUS => "Data_Modbus_RTU_Ro".Modbus_Master.Status)
   END_RUNG
   // the same network as SCL:
   "Modbus_RTU_V1.0_DB_Lift"(PORT := "Local~CM_1241_(RS422_485)_1",   // "Modbus_RTU_V1.0_Lift"
                           BAUD := 115200,
                           Modbus_RTU_ADDR := "Data_Modbus_RTU_Lift".Address_INVT,
                           MODE := 1,
                           MODE_1 := 0,
                           DATA_LEN := 1,
                           Modbus_Master_DONE := "Data_Modbus_RTU_Lift".Modbus_Master.Done,
                           Modbus_Master_ERROR := "Data_Modbus_RTU_Lift".Modbus_Master.Error,
                           "Step" := "Data_Modbus_RTU_Lift"."Step",
                           Req_Comm_Load := "Data_Modbus_RTU_Lift"."Modbus_Comm_Load-".Req,
                           Req_Modbus_Master := "Data_Modbus_RTU_Lift".Modbus_Master.Req,
                           ADDR_Resistor_Startus := "Data_Modbus_RTU_Lift".Address_Status,
                           ADDR_Resistor_Speed := "Data_Modbus_RTU_Lift".Address_Speed,
                           ADDR_Resistor_Current_HZ_Volt := "Data_Modbus_RTU_Lift".Address_Current_HZ_Volt,
                           Data_Run_INVT := "Data_Control".Elevator.DataSTATUSControl_INVT,
                           Data_Speed := "Data_Control".Elevator.DataSPEEDLift_INVT,
                           data_Mb := "Data_mb_E".Data_Mb,
                           Done_Comm_Load => "Data_Modbus_RTU_Lift"."Modbus_Comm_Load-".Done,
                           Error_Comm_Load => "Data_Modbus_RTU_Lift"."Modbus_Comm_Load-".Error,
                           STATUS_Comm_Load => "Data_Modbus_RTU_Lift"."Modbus_Comm_Load-".Status,
                           Modbus_Master_BUSY => "Data_Modbus_RTU_Lift".Modbus_Master.Busy,
                           Modbus_Master_STATUS => "Data_Modbus_RTU_Lift".Modbus_Master.Status);
   "Modbus_RTU_V1.0_Tray_DB"(PORT := "Local~CM_1241_(RS422_485)_3",   // "Modbus_RTU_V1.0_Tray"
                           BAUD := 38400,
                           Modbus_RTU_ADDR := "Data_Modbus_RTU_Tray".Address_INVT,
                           MODE := 1,
                           MODE_1 := 0,
                           DATA_LEN := 1,
                           Modbus_Master_ERROR := "Data_Modbus_RTU_Tray".Modbus_Master.Error,
                           Modbus_Master_DONE := "Data_Modbus_RTU_Tray".Modbus_Master.Done,
                           "Step" := "Data_Modbus_RTU_Tray"."Step",
                           Req_Comm_Load := "Data_Modbus_RTU_Tray"."Modbus_Comm_Load-".Req,
                           Req_Modbus_Master := "Data_Modbus_RTU_Tray".Modbus_Master.Req,
                           ADDR_Resistor_Startus := "Data_Modbus_RTU_Tray".Address_Status,
                           ADDR_Resistor_Speed := "Data_Modbus_RTU_Tray".Address_Speed,
                           ADDR_Resistor_Current_HZ_Volt := "Data_Modbus_RTU_Tray".ADDR_Resistor_Current_HZ_Volt,
                           MB_DB := "Modbus_Master_DB_1".MB_DB,
                           Data_Run_INVT := "Data_Control".HookPallet.DataSTATUSControl_INVT,
                           Data_Speed := "Data_Control".HookPallet.DataSPEEDLift_INVT,
                           data_mb := "Data_mb_T".Data_Mb,
                           Done_Comm_Load => "Data_Modbus_RTU_Tray"."Modbus_Comm_Load-".Done,
                           Error_Comm_Load => "Data_Modbus_RTU_Tray"."Modbus_Comm_Load-".Error,
                           STATUS_Comm_Load => "Data_Modbus_RTU_Tray"."Modbus_Comm_Load-".Status,
                           Modbus_Master_BUSY => "Data_Modbus_RTU_Tray".Modbus_Master.Busy,
                           Modbus_Master_STATUS => "Data_Modbus_RTU_Tray".Modbus_Master.Status);
   "Modbus_RTU_V1.0_Ro_DB"(PORT := "Local~CM_1241_(RS422_485)_2",   // "Modbus_RTU_V1.0_Ro"
                           BAUD := 38400,
                           Modbus_RTU_ADDR := "Data_Modbus_RTU_Ro".Address_INVT,
                           MODE := 1,
                           MODE_1 := 0,
                           DATA_LEN := 1,
                           Modbus_Master_DONE := "Data_Modbus_RTU_Ro".Modbus_Master.Done,
                           Modbus_Master_ERROR := "Data_Modbus_RTU_Ro".Modbus_Master.Error,
                           "Step" := "Data_Modbus_RTU_Ro"."Step",
                           Req_Comm_Load := "Data_Modbus_RTU_Ro"."Modbus_Comm_Load-".Req,
                           Req_Modbus_Master := "Data_Modbus_RTU_Ro".Modbus_Master.Req,
                           ADDR_Resistor_Startus := "Data_Modbus_RTU_Ro".Address_Status,
                           ADDR_Resistor_Current := "Data_Modbus_RTU_Ro".Address_Current_HZ_Volt,
                           ADDR_Resistor_Speed := "Data_Modbus_RTU_Ro".Address_Speed,
                           MB_DB := "Modbus_Master_DB_2".MB_DB,
                           Data_Run_INVT := "Data_Control".TableRotation.DataStatusINVT,
                           Data_Speed := "Data_Control".TableRotation.DataSpeedINVT,
                           Data_MB := "Data_MB_R".Data_Mb,
                           Done_Comm_Load => "Data_Modbus_RTU_Ro"."Modbus_Comm_Load-".Done,
                           Error_Comm_Load => "Data_Modbus_RTU_Ro"."Modbus_Comm_Load-".Error,
                           STATUS_Comm_Load => "Data_Modbus_RTU_Ro"."Modbus_Comm_Load-".Status,
                           Modbus_Master_BUSY => "Data_Modbus_RTU_Ro".Modbus_Master.Busy,
                           Modbus_Master_STATUS => "Data_Modbus_RTU_Ro".Modbus_Master.Status);
END_REGION
END_FUNCTION_BLOCK

// folder: Control/Modbus RTU/Modbus RTU_Lift

FUNCTION_BLOCK "Modbus_RTU_V1.0_Lift"   // FB1, LAD
{ S7_Optimized_Access := 'FALSE' }
VERSION : 0.1
   VAR_INPUT
      PORT : Port;
      BAUD : UDInt;
      Modbus_RTU_ADDR : UInt;   // Modbus RTU Stationsadresse
      MODE : USInt;   // Bezeichnet die Art der Anforderung
      MODE_1 : USInt := 1;
      DATA_LEN : UInt;   // Datenlänge: Anzahl der Bits oder Wörter
   END_VAR
   VAR_OUTPUT
      Done_Comm_Load : Bool;
      Error_Comm_Load : Bool;
      STATUS_Comm_Load : Word;
      Modbus_Master_BUSY : Bool;
      Modbus_Master_STATUS : Word;
   END_VAR
   VAR_IN_OUT
      Modbus_Master_DONE : Bool;
      Modbus_Master_ERROR : Bool;
      "Step" : Int;
      Req_Comm_Load : Bool;
      Req_Modbus_Master : Bool;
      ADDR_Resistor_Startus : UInt;   // Anfangsadresse im Slave
      ADDR_Resistor_Speed : UInt;
      ADDR_Resistor_Current_HZ_Volt : UInt;
      Data_Run_INVT : Word;
      Data_Speed : Int;
      data_Mb : Struct
         Data_HZ : Int;
         Data_Current : Int;
         Data_Volt : Int;
      END_STRUCT;
   END_VAR
   VAR_TEMP   // added for the SCL form of the ladder/FBD networks
      _w1 : Bool;
   END_VAR
BEGIN

REGION Network 1
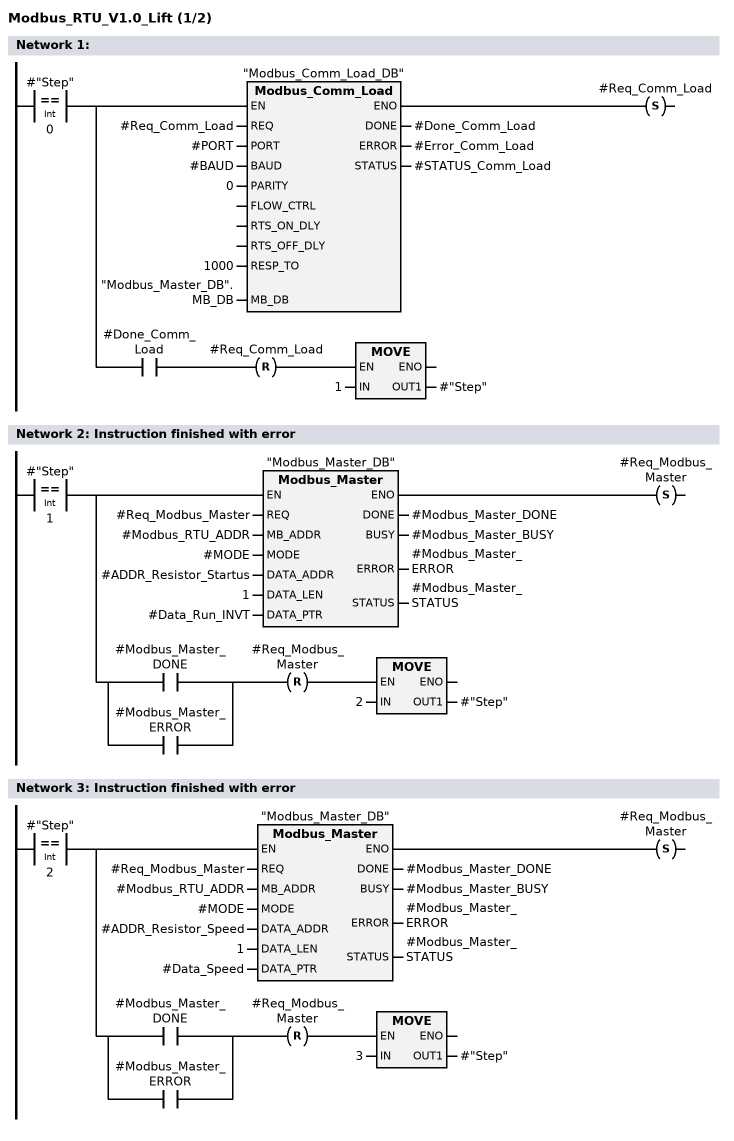
   // ENO of a box is taken as its EN; it also drops when the box reports an error
   #_w1 := #"Step" = 0;
   IF #_w1 THEN
       "Modbus_Comm_Load_DB"(REQ := #Req_Comm_Load,   // Modbus_Comm_Load
                             PORT := #PORT,
                             BAUD := #BAUD,
                             PARITY := 0,
                             RESP_TO := 1000,
                             MB_DB := "Modbus_Master_DB".MB_DB,
                             DONE => #Done_Comm_Load,
                             ERROR => #Error_Comm_Load,
                             STATUS => #STATUS_Comm_Load);
       #Req_Comm_Load := TRUE;
   END_IF;
   IF #_w1 AND #Done_Comm_Load THEN
       #Req_Comm_Load := FALSE;
       #"Step" := 1;
   END_IF;
END_REGION

REGION Network 2: Instruction finished with error
   // ENO of a box is taken as its EN; it also drops when the box reports an error
   #_w1 := #"Step" = 1;
   IF #_w1 THEN
       "Modbus_Master_DB"(REQ := #Req_Modbus_Master,   // Modbus_Master
                          MB_ADDR := #Modbus_RTU_ADDR,
                          MODE := #MODE,
                          DATA_ADDR := #ADDR_Resistor_Startus,
                          DATA_LEN := 1,
                          DATA_PTR := #Data_Run_INVT,
                          DONE => #Modbus_Master_DONE,
                          BUSY => #Modbus_Master_BUSY,
                          ERROR => #Modbus_Master_ERROR,
                          STATUS => #Modbus_Master_STATUS);
       #Req_Modbus_Master := TRUE;
   END_IF;
   IF #_w1 AND (#Modbus_Master_DONE OR #Modbus_Master_ERROR) THEN
       #Req_Modbus_Master := FALSE;
       #"Step" := 2;
   END_IF;
END_REGION

REGION Network 3: Instruction finished with error
   // ENO of a box is taken as its EN; it also drops when the box reports an error
   #_w1 := #"Step" = 2;
   IF #_w1 THEN
       "Modbus_Master_DB"(REQ := #Req_Modbus_Master,   // Modbus_Master
                          MB_ADDR := #Modbus_RTU_ADDR,
                          MODE := #MODE,
                          DATA_ADDR := #ADDR_Resistor_Speed,
                          DATA_LEN := 1,
                          DATA_PTR := #Data_Speed,
                          DONE => #Modbus_Master_DONE,
                          BUSY => #Modbus_Master_BUSY,
                          ERROR => #Modbus_Master_ERROR,
                          STATUS => #Modbus_Master_STATUS);
       #Req_Modbus_Master := TRUE;
   END_IF;
   IF #_w1 AND (#Modbus_Master_DONE OR #Modbus_Master_ERROR) THEN
       #Req_Modbus_Master := FALSE;
       #"Step" := 3;
   END_IF;
END_REGION

REGION Network 4: Instruction finished with error
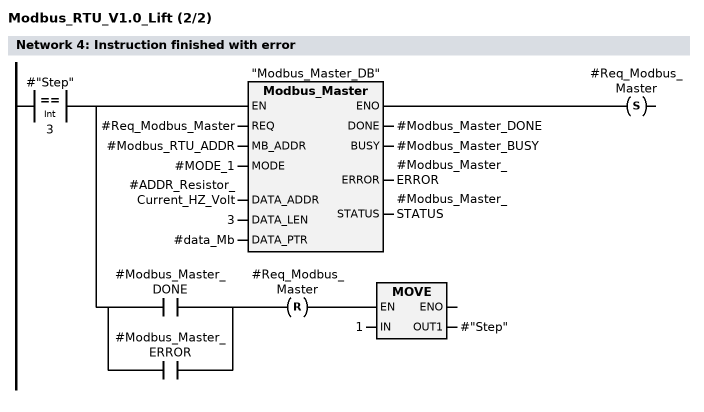
   // ENO of a box is taken as its EN; it also drops when the box reports an error
   #_w1 := #"Step" = 3;
   IF #_w1 THEN
       "Modbus_Master_DB"(REQ := #Req_Modbus_Master,   // Modbus_Master
                          MB_ADDR := #Modbus_RTU_ADDR,
                          MODE := #MODE_1,
                          DATA_ADDR := #ADDR_Resistor_Current_HZ_Volt,
                          DATA_LEN := 3,
                          DATA_PTR := #data_Mb,
                          DONE => #Modbus_Master_DONE,
                          BUSY => #Modbus_Master_BUSY,
                          ERROR => #Modbus_Master_ERROR,
                          STATUS => #Modbus_Master_STATUS);
       #Req_Modbus_Master := TRUE;
   END_IF;
   IF #_w1 AND (#Modbus_Master_DONE OR #Modbus_Master_ERROR) THEN
       #Req_Modbus_Master := FALSE;
       #"Step" := 1;
   END_IF;
END_REGION
END_FUNCTION_BLOCK

// folder: Control/Modbus RTU/Modbus_RTU_Ro

FUNCTION_BLOCK "Modbus_RTU_V1.0_Ro"   // FB9, LAD
{ S7_Optimized_Access := 'FALSE' }
VERSION : 0.1
   VAR_INPUT
      PORT : Port;
      BAUD : UDInt;
      Modbus_RTU_ADDR : UInt;   // Modbus RTU Stationsadresse
      MODE : USInt;   // Bezeichnet die Art der Anforderung
      MODE_1 : USInt := 1;
      DATA_LEN : UInt;   // Datenlänge: Anzahl der Bits oder Wörter
   END_VAR
   VAR_OUTPUT
      Done_Comm_Load : Bool;
      Error_Comm_Load : Bool;
      STATUS_Comm_Load : Word;
      Modbus_Master_BUSY : Bool;
      Modbus_Master_STATUS : Word;
   END_VAR
   VAR_IN_OUT
      Modbus_Master_DONE : Bool;
      Modbus_Master_ERROR : Bool;
      "Step" : Int;
      Req_Comm_Load : Bool;
      Req_Modbus_Master : Bool;
      ADDR_Resistor_Startus : UInt;   // Anfangsadresse im Slave
      ADDR_Resistor_Current : UInt;
      ADDR_Resistor_Speed : UInt;
      MB_DB : P2P_MB_BASE;   // Modbus Parameter / Modbus parameters
      Data_Run_INVT : Word;
      Data_Speed : Int;
      Data_MB : Struct
         Data_HZ : Int;
         Data_Current : Int;
         Data_Volt : Int;
      END_STRUCT;
   END_VAR
   VAR_TEMP   // added for the SCL form of the ladder/FBD networks
      _w1 : Bool;
   END_VAR
BEGIN

REGION Network 1
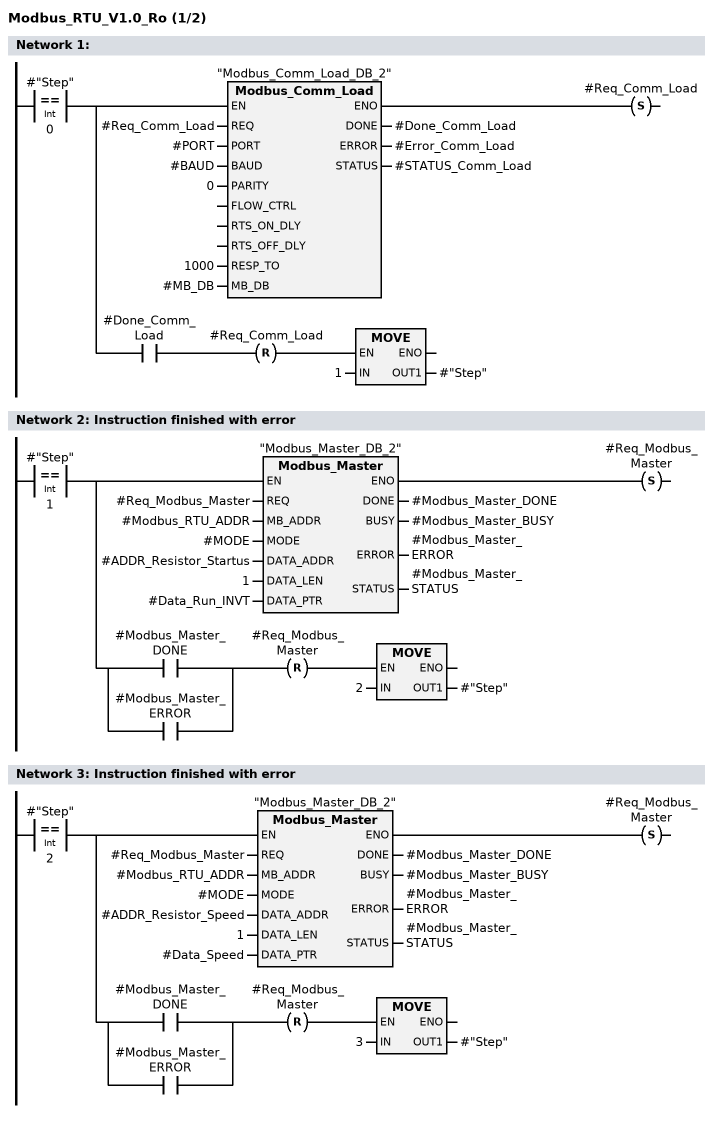
   // ENO of a box is taken as its EN; it also drops when the box reports an error
   #_w1 := #"Step" = 0;
   IF #_w1 THEN
       "Modbus_Comm_Load_DB_2"(REQ := #Req_Comm_Load,   // Modbus_Comm_Load
                               PORT := #PORT,
                               BAUD := #BAUD,
                               PARITY := 0,
                               RESP_TO := 1000,
                               MB_DB := #MB_DB,
                               DONE => #Done_Comm_Load,
                               ERROR => #Error_Comm_Load,
                               STATUS => #STATUS_Comm_Load);
       #Req_Comm_Load := TRUE;
   END_IF;
   IF #_w1 AND #Done_Comm_Load THEN
       #Req_Comm_Load := FALSE;
       #"Step" := 1;
   END_IF;
END_REGION

REGION Network 2: Instruction finished with error
   // ENO of a box is taken as its EN; it also drops when the box reports an error
   #_w1 := #"Step" = 1;
   IF #_w1 THEN
       "Modbus_Master_DB_2"(REQ := #Req_Modbus_Master,   // Modbus_Master
                            MB_ADDR := #Modbus_RTU_ADDR,
                            MODE := #MODE,
                            DATA_ADDR := #ADDR_Resistor_Startus,
                            DATA_LEN := 1,
                            DATA_PTR := #Data_Run_INVT,
                            DONE => #Modbus_Master_DONE,
                            BUSY => #Modbus_Master_BUSY,
                            ERROR => #Modbus_Master_ERROR,
                            STATUS => #Modbus_Master_STATUS);
       #Req_Modbus_Master := TRUE;
   END_IF;
   IF #_w1 AND (#Modbus_Master_DONE OR #Modbus_Master_ERROR) THEN
       #Req_Modbus_Master := FALSE;
       #"Step" := 2;
   END_IF;
END_REGION

REGION Network 3: Instruction finished with error
   // ENO of a box is taken as its EN; it also drops when the box reports an error
   #_w1 := #"Step" = 2;
   IF #_w1 THEN
       "Modbus_Master_DB_2"(REQ := #Req_Modbus_Master,   // Modbus_Master
                            MB_ADDR := #Modbus_RTU_ADDR,
                            MODE := #MODE,
                            DATA_ADDR := #ADDR_Resistor_Speed,
                            DATA_LEN := 1,
                            DATA_PTR := #Data_Speed,
                            DONE => #Modbus_Master_DONE,
                            BUSY => #Modbus_Master_BUSY,
                            ERROR => #Modbus_Master_ERROR,
                            STATUS => #Modbus_Master_STATUS);
       #Req_Modbus_Master := TRUE;
   END_IF;
   IF #_w1 AND (#Modbus_Master_DONE OR #Modbus_Master_ERROR) THEN
       #Req_Modbus_Master := FALSE;
       #"Step" := 3;
   END_IF;
END_REGION

REGION Network 4: Instruction finished with error
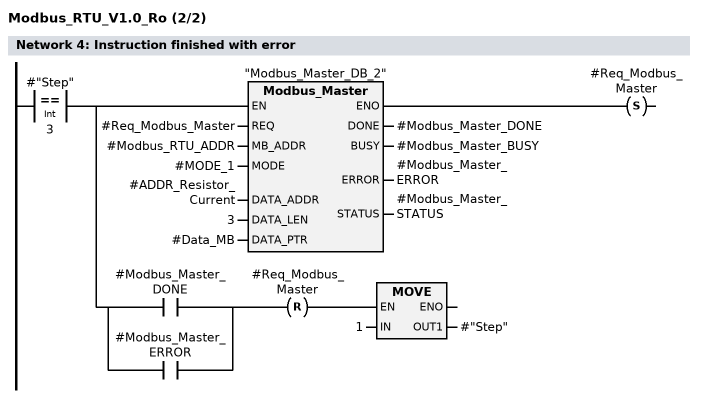
   // ENO of a box is taken as its EN; it also drops when the box reports an error
   #_w1 := #"Step" = 3;
   IF #_w1 THEN
       "Modbus_Master_DB_2"(REQ := #Req_Modbus_Master,   // Modbus_Master
                            MB_ADDR := #Modbus_RTU_ADDR,
                            MODE := #MODE_1,
                            DATA_ADDR := #ADDR_Resistor_Current,
                            DATA_LEN := 3,
                            DATA_PTR := #Data_MB,
                            DONE => #Modbus_Master_DONE,
                            BUSY => #Modbus_Master_BUSY,
                            ERROR => #Modbus_Master_ERROR,
                            STATUS => #Modbus_Master_STATUS);
       #Req_Modbus_Master := TRUE;
   END_IF;
   IF #_w1 AND (#Modbus_Master_DONE OR #Modbus_Master_ERROR) THEN
       #Req_Modbus_Master := FALSE;
       #"Step" := 1;
   END_IF;
END_REGION
END_FUNCTION_BLOCK

// folder: Control/Modbus RTU/Modbus_RTU_Tray

FUNCTION_BLOCK "Modbus_RTU_V1.0_Tray"   // FB10, LAD
{ S7_Optimized_Access := 'FALSE' }
VERSION : 0.1
   VAR_INPUT
      PORT : Port;
      BAUD : UDInt;
      Modbus_RTU_ADDR : UInt;   // Modbus RTU Stationsadresse
      MODE : USInt;   // Bezeichnet die Art der Anforderung
      MODE_1 : USInt;
      DATA_LEN : UInt;   // Datenlänge: Anzahl der Bits oder Wörter
   END_VAR
   VAR_OUTPUT
      Done_Comm_Load : Bool;
      Error_Comm_Load : Bool;
      STATUS_Comm_Load : Word;
      Modbus_Master_BUSY : Bool;
      Modbus_Master_STATUS : Word;
   END_VAR
   VAR_IN_OUT
      Modbus_Master_ERROR : Bool;
      Modbus_Master_DONE : Bool;
      "Step" : Int;
      Req_Comm_Load : Bool;
      Req_Modbus_Master : Bool;
      ADDR_Resistor_Startus : UInt;   // Anfangsadresse im Slave
      ADDR_Resistor_Speed : UInt;
      ADDR_Resistor_Current_HZ_Volt : UInt;
      MB_DB : P2P_MB_BASE;   // Modbus Parameter / Modbus parameters
      Data_Run_INVT : Word;
      Data_Speed : Int;
      data_mb : Struct
         Data_HZ : Int;
         Data_Current : Int;
         Data_Volt : Int;
      END_STRUCT;
   END_VAR
   VAR_TEMP   // added for the SCL form of the ladder/FBD networks
      _w1 : Bool;
   END_VAR
BEGIN

REGION Network 1
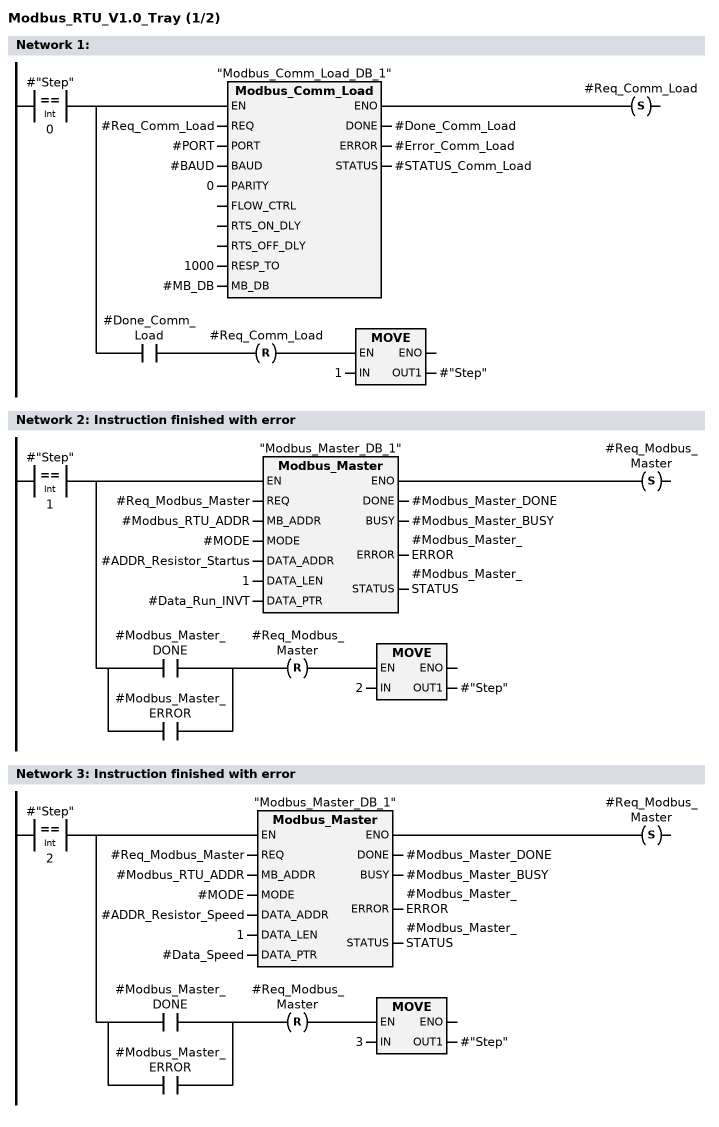
   // ENO of a box is taken as its EN; it also drops when the box reports an error
   #_w1 := #"Step" = 0;
   IF #_w1 THEN
       "Modbus_Comm_Load_DB_1"(REQ := #Req_Comm_Load,   // Modbus_Comm_Load
                               PORT := #PORT,
                               BAUD := #BAUD,
                               PARITY := 0,
                               RESP_TO := 1000,
                               MB_DB := #MB_DB,
                               DONE => #Done_Comm_Load,
                               ERROR => #Error_Comm_Load,
                               STATUS => #STATUS_Comm_Load);
       #Req_Comm_Load := TRUE;
   END_IF;
   IF #_w1 AND #Done_Comm_Load THEN
       #Req_Comm_Load := FALSE;
       #"Step" := 1;
   END_IF;
END_REGION

REGION Network 2: Instruction finished with error
   // ENO of a box is taken as its EN; it also drops when the box reports an error
   #_w1 := #"Step" = 1;
   IF #_w1 THEN
       "Modbus_Master_DB_1"(REQ := #Req_Modbus_Master,   // Modbus_Master
                            MB_ADDR := #Modbus_RTU_ADDR,
                            MODE := #MODE,
                            DATA_ADDR := #ADDR_Resistor_Startus,
                            DATA_LEN := 1,
                            DATA_PTR := #Data_Run_INVT,
                            DONE => #Modbus_Master_DONE,
                            BUSY => #Modbus_Master_BUSY,
                            ERROR => #Modbus_Master_ERROR,
                            STATUS => #Modbus_Master_STATUS);
       #Req_Modbus_Master := TRUE;
   END_IF;
   IF #_w1 AND (#Modbus_Master_DONE OR #Modbus_Master_ERROR) THEN
       #Req_Modbus_Master := FALSE;
       #"Step" := 2;
   END_IF;
END_REGION

REGION Network 3: Instruction finished with error
   // ENO of a box is taken as its EN; it also drops when the box reports an error
   #_w1 := #"Step" = 2;
   IF #_w1 THEN
       "Modbus_Master_DB_1"(REQ := #Req_Modbus_Master,   // Modbus_Master
                            MB_ADDR := #Modbus_RTU_ADDR,
                            MODE := #MODE,
                            DATA_ADDR := #ADDR_Resistor_Speed,
                            DATA_LEN := 1,
                            DATA_PTR := #Data_Speed,
                            DONE => #Modbus_Master_DONE,
                            BUSY => #Modbus_Master_BUSY,
                            ERROR => #Modbus_Master_ERROR,
                            STATUS => #Modbus_Master_STATUS);
       #Req_Modbus_Master := TRUE;
   END_IF;
   IF #_w1 AND (#Modbus_Master_DONE OR #Modbus_Master_ERROR) THEN
       #Req_Modbus_Master := FALSE;
       #"Step" := 3;
   END_IF;
END_REGION

REGION Network 4: Instruction finished with error
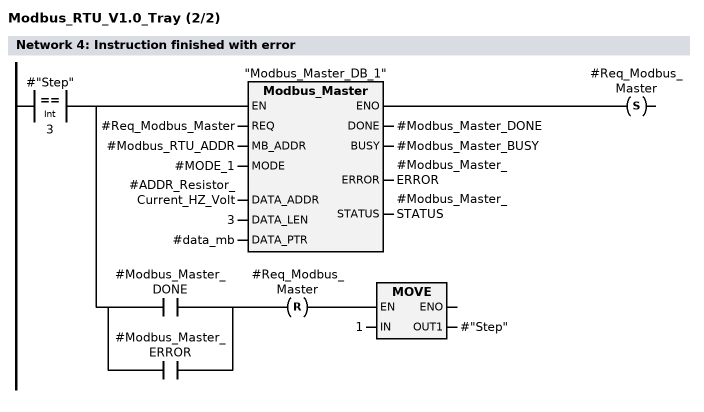
   // ENO of a box is taken as its EN; it also drops when the box reports an error
   #_w1 := #"Step" = 3;
   IF #_w1 THEN
       "Modbus_Master_DB_1"(REQ := #Req_Modbus_Master,   // Modbus_Master
                            MB_ADDR := #Modbus_RTU_ADDR,
                            MODE := #MODE_1,
                            DATA_ADDR := #ADDR_Resistor_Current_HZ_Volt,
                            DATA_LEN := 3,
                            DATA_PTR := #data_mb,
                            DONE => #Modbus_Master_DONE,
                            BUSY => #Modbus_Master_BUSY,
                            ERROR => #Modbus_Master_ERROR,
                            STATUS => #Modbus_Master_STATUS);
       #Req_Modbus_Master := TRUE;
   END_IF;
   IF #_w1 AND (#Modbus_Master_DONE OR #Modbus_Master_ERROR) THEN
       #Req_Modbus_Master := FALSE;
       #"Step" := 1;
   END_IF;
END_REGION
END_FUNCTION_BLOCK

(* ===== HMI "HMI_RT_1" =====
system functions are stored by id; their names below are inferred from use
connection "HMI_Connection_1": ETHERNET, SMART_S7_1200_OMS

HMI tags "Default tag table"
   "Data_Control_Elevator_FloorAddressReal" : Int = PLC Data_Control.Elevator.FloorAddressReal AT %DB5.DBW52, 1 s
   "Data_Control_SlotIDFrom" : Int = PLC Data_Control.SlotIDFrom AT %DB5.DBW18, 1 s
   "Data_Control_SlotIDTO" : Int = PLC Data_Control.SlotIDTO AT %DB5.DBW20, 1 s
   "Data_Control_ERROR" : Bool = PLC Data_Control.ERROR AT %DB5.DBX10.6, 1 s
   "Data_Control_ModeAction" : Int = PLC Data_Control.ModeAction AT %DB5.DBW14, 1 s
   "Data_Control_Elevator_DataSPEEDLift_INVT" : Int = PLC Data_Control.Elevator.DataSPEEDLift_INVT AT %DB5.DBW40, 1 s
   "Data_Control_HookPallet_DataSPEEDLift_INVT" : Int = PLC Data_Control.HookPallet.DataSPEEDLift_INVT AT %DB5.DBW112, 1 s
   "Data_Control_TableRotation_DataSpeedINVT" : Int = PLC Data_Control.TableRotation.DataSpeedINVT AT %DB5.DBW184, 1 s
   "Data_Control_Elevator_Running" : Bool = PLC Data_Control.Elevator.Running AT %DB5.DBX26.2, 1 s
   "Data_Control_HookPallet_Running" : Bool = PLC Data_Control.HookPallet.Running AT %DB5.DBX70.2, 1 s
   "Data_Control_Stop" : Bool = PLC Data_Control.Stop AT %DB5.DBX10.0, 1 s
   "Data_Control_Elevator_UP" : Bool = PLC Data_Control.Elevator.UP AT %DB5.DBX26.4, 1 s
   "Data_Control_Elevator_DOWN" : Bool = PLC Data_Control.Elevator.DOWN AT %DB5.DBX26.5, 1 s
   "Data_Control_HookPallet_1" : Bool = PLC Data_Control.HookPallet.1 AT %DB5.DBX70.3, 1 s
   "Data_Control_HookPallet_2" : Bool = PLC Data_Control.HookPallet.2 AT %DB5.DBX70.4, 1 s
   "Data_Control_TableRotation_Up_Manual" : Bool = PLC Data_Control.TableRotation.Up_Manual AT %DB5.DBX182.0, 1 s
   "Data_Control_TableRotation_Down_Manual" : Bool = PLC Data_Control.TableRotation.Down_Manual AT %DB5.DBX182.1, 1 s
   "Data_Control_TableRotation_Ro.1_Manual" : Bool = PLC Data_Control.TableRotation."Ro.1_Manual" AT %DB5.DBX182.2, 1 s
   "Data_Control_TableRotation_Ro.2_Manual" : Bool = PLC Data_Control.TableRotation."Ro.2_Manual" AT %DB5.DBX182.3, 1 s
   "Data_ADMIN_HMI_Position_201" : Bool = PLC Data_ADMIN_HMI.Position.201 AT %DB26.DBX2.0, 1 s
   "Data_ADMIN_HMI_Position_202" : Bool = PLC Data_ADMIN_HMI.Position.202 AT %DB26.DBX2.1, 1 s
   "Data_ADMIN_HMI_PositionNumber" : Int = PLC Data_ADMIN_HMI.PositionNumber AT %DB26.DBW6, 1 s
   "Data_ADMIN_HMI_OKE" : Bool = PLC Data_ADMIN_HMI.OKE AT %DB26.DBX0.0, 1 s
   "Data_Control_ModeNumber" : Int = PLC Data_Control.ModeNumber AT %DB5.DBW16, 1 s
   "Data_Control_Auto_Manual" : Bool = PLC Data_Control.Auto_Manual AT %DB5.DBX10.3, 1 s
   "Data_Control_Auto.Mode2_Mode1" : Bool = PLC Data_Control."Auto.Mode2_Mode1" AT %DB5.DBX10.5, 1 s
   "Data_Control_Auto.Mode1_Mode2" : Bool = PLC Data_Control."Auto.Mode1_Mode2" AT %DB5.DBX10.4, 1 s
   "Data_ADMIN_HMI_Position_101" : Bool = PLC Data_ADMIN_HMI.Position.101 AT %DB26.DBX2.2, 1 s
   "Data_ADMIN_HMI_Position_102" : Bool = PLC Data_ADMIN_HMI.Position.102 AT %DB26.DBX2.3, 1 s
   "Data_ADMIN_HMI_CheckPosition_101" : Bool = PLC Data_ADMIN_HMI.CheckPosition.101 AT %DB26.DBX4.2, 1 s
   "Data_ADMIN_HMI_CheckPosition_102" : Bool = PLC Data_ADMIN_HMI.CheckPosition.102 AT %DB26.DBX4.3, 1 s
   "Data_ADMIN_HMI_CheckPosition_201" : Bool = PLC Data_ADMIN_HMI.CheckPosition.201 AT %DB26.DBX4.0, 1 s
   "Data_ADMIN_HMI_CheckPosition_202" : Bool = PLC Data_ADMIN_HMI.CheckPosition.202 AT %DB26.DBX4.1, 1 s
   "Data_Control_RST" : Bool = PLC Data_Control.RST AT %DB5.DBX10.2, 1 s
   "Data_Control_START" : Bool = PLC Data_Control.START AT %DB5.DBX10.1, 1 s
   "Data_Control_ERRORNumber" : Int = PLC Data_Control.ERRORNumber AT %DB5.DBW12, 1 s
   "Data_Control_Auto.Mode1_Elevator" : Bool = PLC Data_Control."Auto.ACTION".Elevator AT %DB5.DBX24.0, 1 s
   "Data_Control_Auto.Mode1_HookPallet" : Bool = PLC Data_Control."Auto.ACTION".HookPallet AT %DB5.DBX24.2, 1 s
   "Data_Control_Auto.Mode1_TableRotation" : Bool = PLC Data_Control."Auto.ACTION".TableRotation AT %DB5.DBX24.4, 1 s
   "Data_ADMIN_HMI_blink" : Bool = PLC Data_ADMIN_HMI.blink_Manual AT %DB26.DBX0.1, 1 s
   "Data_ADMIN_HMI_blink_Setup" : Bool = PLC Data_ADMIN_HMI.blink_Setup AT %DB26.DBX0.4, 1 s
   "Data_ADMIN_HMI_blink_Back" : Bool = PLC Data_ADMIN_HMI.blink_Back AT %DB26.DBX0.5, 1 s
   "Data_ADMIN_HMI_blink_Position" : Bool = PLC Data_ADMIN_HMI.blink_Position AT %DB26.DBX0.6, 1 s
   "Data_ADMIN_HMI_blink_Cancel" : Bool = PLC Data_ADMIN_HMI.blink_Cancel AT %DB26.DBX0.3, 1 s
   "Data_ADMIN_HMI_blink_Auto" : Bool = PLC Data_ADMIN_HMI.blink_Auto AT %DB26.DBX0.2, 1 s
   "SS01" : Bool = PLC SS01 AT %I0.1, 1 s
   "SS00" : Bool = PLC SS00 AT %I0.0, 1 s
   "SS13" : Bool = PLC SS13 AT %I1.5, 1 s
   "SS12" : Bool = PLC SS12 AT %I1.4, 1 s
   "SS07" : Bool = PLC SS07 AT %I0.7, 1 s
   "SS08" : Bool = PLC SS08 AT %I1.0, 1 s
   "SS04" : Bool = PLC SS04 AT %I0.4, 1 s
   "SS03" : Bool = PLC SS03 AT %I0.3, 1 s

screen "Root screen" 800x480
   TextField "Text field_1" at 271,53 size 257x32; Text 'ATOMA TECHNOLOGY'
   TextField "Text field_4" at 175,10 size 443x43; Text 'ATOMA PARKING SYSTEMS'
   Button "Button_1" at 0,417 size 222x63; TextOff 'SETUP'
      on Click: ActivateScreen("SETUP", 0)
      on Press: SetBit("Data_ADMIN_HMI_blink_Setup")
      on Release: ResetBit("Data_ADMIN_HMI_blink_Setup")
      Appearance <- "Data_ADMIN_HMI_blink_Setup"
   Button "Button_2" at 223,417 size 222x63; TextOff 'MANUAL'
      on Click: ActivateScreen("MANUAL", 0)
      Appearance <- "Data_ADMIN_HMI_blink"
      on Release: ResetBit("Data_ADMIN_HMI_blink")
      on Press: SetBit("Data_ADMIN_HMI_blink")
   Button "Button_3" at 446,416 size 222x63; TextOff 'AUTO'
      on Click: ActivateScreen("AUTO", 0)
      on Press: SetBit("Data_ADMIN_HMI_blink_Auto")
      on Release: ResetBit("Data_ADMIN_HMI_blink_Auto")
      Appearance <- "Data_ADMIN_HMI_blink_Auto"
   Button "Button_4" at 669,203 size 129x276; TextOff 'STOP'
      on Press: SetBit("Data_Control_Stop")
      on Release: ResetBit("Data_Control_Stop")
      Appearance <- "Data_Control_Stop"
   IOField "I/O field_2" at 18,133 size 106x41; FormatPattern s999
      ProcessValue <- "Data_Control_SlotIDFrom"
   TextField "Text field_3" at 39,178 size 50x22; Text 'FROM'
   IOField "I/O field_3" at 466,133 size 106x41; FormatPattern 1
      ProcessValue <- "Data_Control_ERROR"
      Appearance <- "Data_Control_ERROR"
   TextField "Text field_2" at 489,178 size 63x22; Text 'ERROR'
   IOField "I/O field_1" at 683,133 size 106x41; FormatPattern s999
      ProcessValue <- "Data_Control_ModeNumber"
   TextField "Text field_8" at 680,178 size 114x22; Text 'MODE ACTION'
   Circle "Circle_1" at 59,262 size 48x48
      Appearance <- "Data_Control_Elevator_Running"
   IOField "I/O field_4" at 33,327 size 96x32; FormatPattern s99999
      ProcessValue <- "Data_Control_Elevator_DataSPEEDLift_INVT"
   IOField "I/O field_5" at 206,327 size 96x32; FormatPattern s99999
      ProcessValue <- "Data_Control_TableRotation_DataSpeedINVT"
   Circle "Circle_3" at 416,262 size 48x48
      Appearance <- "Data_Control_HookPallet_Running"
   IOField "I/O field_6" at 393,327 size 96x32; FormatPattern s99999
      ProcessValue <- "Data_Control_HookPallet_DataSPEEDLift_INVT"
   IOField "I/O field_7" at 554,327 size 96x32; FormatPattern 9999999
   IOField "I/O field_8" at 242,133 size 106x41; FormatPattern s999
      ProcessValue <- "Data_Control_SlotIDTO"
   TextField "Text field_9" at 273,178 size 38x22; Text 'TO'
   TextField "Text field_10" at 155,144 size 44x23; Text '==>'
   TextField "Text field_11" at 45,230 size 92x23; Text 'ELEVATOR'
   TextField "Text field_12" at 186,230 size 146x23; Text 'TURNING TABLE'
   TextField "Text field_13" at 381,230 size 118x23; Text 'TRAY PALLET'
   TextField "Text field_14" at 576,230 size 51x23; Text 'DONE'
   IOField "I/O field_9" at 555,378 size 96x32; FormatPattern 9999999
   TextField "Text field_15" at 138,175 size 70x23; Text '====>'

screen "SETUP" 800x480
   Button "Button_1" at 1,421 size 113x58; TextOff 'BACK'; TextOn 'Root screen'
      on Click: ActivateScreen("Root screen", 0)
      on Press: SetBit("Data_ADMIN_HMI_blink_Back")
      on Release: ResetBit("Data_ADMIN_HMI_blink_Back")
      Appearance <- "Data_ADMIN_HMI_blink_Back"
   Switch "Switch_2" at 507,338 size 287x62; TextOn 'AUTO MODE 2'; CaptionText 'Switch'; TextOff 'AUTO MODE 1'
      ProcessValue <- "Data_Control_Auto.Mode1_Mode2"
   IOField "I/O field_1" at 643,120 size 140x43; FormatPattern s99999
      ProcessValue <- "Data_Control_ModeNumber"
   TextField "Text field_2" at 508,130 size 88x23; Text 'MODE ID :'
   IOField "I/O field_2" at 692,2 size 106x41; FormatPattern s99999
      ProcessValue <- "Data_Control_Elevator_FloorAddressReal"
   TextField "Text field_3" at 604,10 size 70x23; Text 'FLOOR :'
   IOField "I/O field_3" at 692,48 size 106x41; FormatPattern s99999
      ProcessValue <- "Data_Control_ERRORNumber"
   TextField "Text field_4" at 604,56 size 74x23; Text 'ERROR :'
   TextField "Text field_5" at 120,177 size 363x27; Text 'Select a Module to control of MODE 1'
   Switch "Switch_4" at 157,236 size 287x65; TextOn 'Elevator'; CaptionText 'Switch'; TextOff 'OFF Elevator'
      ProcessValue <- "Data_Control_Auto.Mode1_Elevator"
   Switch "Switch_5" at 157,314 size 287x62; TextOn 'Hook Pallet'; CaptionText 'Switch'; TextOff 'Off HP'
      ProcessValue <- "Data_Control_Auto.Mode1_HookPallet"
   Switch "Switch_6" at 157,389 size 287x62; TextOn 'Table Rotation'; CaptionText 'Switch'; TextOff 'Off TR'
      ProcessValue <- "Data_Control_Auto.Mode1_TableRotation"
   Switch "Switch_1" at 507,204 size 287x65; CaptionText 'Switch'; TextOff 'MANUAL'; TextOn 'AUTO'
      ProcessValue <- "Data_Control_Auto_Manual"
   TextField "Text field_1" at 137,101 size 122x39; Text 'MODE :'

screen "MANUAL" 800x480
   Button "Button_1" at 1,421 size 113x58; TextOn 'Root screen'; TextOff 'BACK'
      on Click: ActivateScreen("Root screen", 0)
      on Press: SetBit("Data_ADMIN_HMI_blink_Back")
      on Release: ResetBit("Data_ADMIN_HMI_blink_Back")
      Appearance <- "Data_ADMIN_HMI_blink_Back"
   Button "Button_2" at 145,146 size 106x66; TextOff 'UP'
      on Release: ResetBit("Data_Control_Elevator_UP")
      on Press: SetBit("Data_Control_Elevator_UP")
      Appearance <- "Data_Control_Elevator_UP"
   Button "Button_3" at 145,307 size 106x66; TextOff 'DOWN'
      on Press: SetBit("Data_Control_Elevator_DOWN")
      on Release: ResetBit("Data_Control_Elevator_DOWN")
      Appearance <- "Data_Control_Elevator_DOWN"
   Button "Button_4" at 278,228 size 106x66; TextOff '2'
      on Press: SetBit("Data_Control_HookPallet_2")
      on Release: ResetBit("Data_Control_HookPallet_2")
      Appearance <- "Data_Control_HookPallet_2"
   Button "Button_5" at 19,227 size 106x66; TextOff '1'
      on Release: ResetBit("Data_Control_HookPallet_1")
      on Press: SetBit("Data_Control_HookPallet_1")
      Appearance <- "Data_Control_HookPallet_1"
   Button "Button_6" at 551,149 size 106x66; TextOff 'UP'
      on Release: ResetBit("Data_Control_TableRotation_Up_Manual")
      on Press: SetBit("Data_Control_TableRotation_Up_Manual")
      Appearance <- "Data_Control_TableRotation_Up_Manual"
   Button "Button_7" at 553,309 size 106x66; TextOff 'DOWN'
      on Press: SetBit("Data_Control_TableRotation_Down_Manual")
      on Release: ResetBit("Data_Control_TableRotation_Down_Manual")
      Appearance <- "Data_Control_TableRotation_Down_Manual"
   Button "Button_8" at 674,230 size 106x66; TextOff 'F'
      on Press: SetBit("Data_Control_TableRotation_Ro.2_Manual")
      on Release: ResetBit("Data_Control_TableRotation_Ro.2_Manual")
      Appearance <- "Data_Control_TableRotation_Ro.2_Manual"
   Button "Button_9" at 418,228 size 106x66; TextOff 'R'
      on Release: ResetBit("Data_Control_TableRotation_Ro.1_Manual")
      on Press: SetBit("Data_Control_TableRotation_Ro.1_Manual")
      Appearance <- "Data_Control_TableRotation_Ro.1_Manual"
   Circle "Circle_1" at 180,217 size 23x23
      Appearance <- "SS04"
   Circle "Circle_2" at 180,281 size 23x23
      Appearance <- "SS03"
   Circle "Circle_3" at 123,249 size 23x23
      Appearance <- "SS07"
   Circle "Circle_4" at 245,249 size 23x23
      Appearance <- "SS08"
   Circle "Circle_5" at 583,220 size 23x23
      Appearance <- "SS01"
   Circle "Circle_6" at 586,284 size 23x23
      Appearance <- "SS00"
   Circle "Circle_7" at 525,252 size 23x23
      Appearance <- "SS12"
   Circle "Circle_8" at 648,252 size 23x23
      Appearance <- "SS13"
   Button "Button_10" at 398,420 size 401x60; TextOn 'AUTO'; TextOff 'AUTO'
      on Click: ActivateScreen("AUTO", 0)
      on Press: SetBit("Data_ADMIN_HMI_blink_Auto")
      on Release: ResetBit("Data_ADMIN_HMI_blink_Auto")
      Appearance <- "Data_ADMIN_HMI_blink_Auto"
   Button "Button_11" at 115,421 size 283x59; TextOn 'SETUP'; TextOff 'SETUP'
      on Click: ActivateScreen("SETUP", 0)
      on Release: ResetBit("Data_ADMIN_HMI_blink_Setup")
      on Press: SetBit("Data_ADMIN_HMI_blink_Setup")
      Appearance <- "Data_ADMIN_HMI_blink_Setup"
   TextField "Text field_11" at 134,11 size 127x32; Text 'ELEVATOR'
   TextField "Text field_12" at 510,6 size 204x32; Text 'TURNING TABLE'
   Circle "Circle_9" at 373,11 size 48x48
      Appearance <- "Data_Control_ERROR"
   IOField "I/O field_4" at 18,89 size 96x32; FormatPattern s99999
      ProcessValue <- "Data_Control_Elevator_DataSPEEDLift_INVT"
   IOField "I/O field_6" at 554,59 size 96x32; FormatPattern s99999
      ProcessValue <- "Data_Control_TableRotation_DataSpeedINVT"
   IOField "I/O field_5" at 281,89 size 96x32; FormatPattern s99999
      ProcessValue <- "Data_Control_HookPallet_DataSPEEDLift_INVT"
   Softkey "Softkey_F3" at 0,0 size 0x0
      on KeyDown: ActivateScreen("AUTO", 0)

screen "AUTO" 800x480
   Button "Button_1" at 1,421 size 134x58; TextOn 'Root screen'; TextOff 'BACK'
      on Click: ActivateScreen("Root screen", 0)
      on Release: ResetBit("Data_ADMIN_HMI_blink_Back")
      on Press: SetBit("Data_ADMIN_HMI_blink_Back")
      Appearance <- "Data_ADMIN_HMI_blink_Back"
   Button "Button_2" at 555,216 size 189x78; TextOff 'START'
      on Click: ActivateScreen("Root screen", 0)
      on Press: SetBit("Data_Control_START")
      on Release: ResetBit("Data_Control_START")
      Appearance <- "Data_Control_START"
   Button "Button_4" at 285,172 size 219x180; TextOff 'EMERGENCY STOP'
      on Release: ResetBit("Data_Control_Stop")
      on Press: SetBit("Data_Control_Stop")
      Appearance <- "Data_Control_Stop"
   Button "Button_3" at 41,216 size 189x78; TextOff 'POSITION PARKING'
      on Click: ActivateScreen("POSITION PARKING", 0)
      on Press: SetBit("Data_ADMIN_HMI_blink_Position")
      on Release: ResetBit("Data_ADMIN_HMI_blink_Position")
      Appearance <- "Data_ADMIN_HMI_blink_Position"
   Button "Button_5" at 295,390 size 189x78; TextOff 'RST'
      on Press: SetBit("Data_Control_RST")
      on Release: ResetBit("Data_Control_RST")
      Appearance <- "Data_Control_RST"
   IOField "I/O field_3" at 7,11 size 138x55; FormatPattern s999
      ProcessValue <- "Data_Control_SlotIDFrom"
   TextField "Text field_1" at 55,70 size 62x27; Text 'FROM'
   IOField "I/O field_4" at 433,11 size 138x55; FormatPattern 1
      ProcessValue <- "Data_Control_ERROR"
      Appearance <- "Data_Control_ERROR"
   TextField "Text field_2" at 467,71 size 63x22; Text 'ERROR'
   IOField "I/O field_5" at 646,11 size 138x55; FormatPattern s999
      ProcessValue <- "Data_Control_ModeNumber"
   TextField "Text field_4" at 658,71 size 114x22; Text 'MODE ACTION'
   IOField "I/O field_6" at 220,11 size 138x55; FormatPattern s999
      ProcessValue <- "Data_Control_SlotIDTO"
   TextField "Text field_5" at 289,70 size 47x27; Text 'TO'
   TextField "Text field_6" at 164,28 size 53x27; Text '==>'
   TextField "Text field_7" at 142,69 size 85x27; Text '====>'

screen "POSITION PARKING" 800x480
   Button "Button_1" at 67,351 size 132x63; TextOff 'OKE'
      on Click: ActivateScreen("AUTO", 0)
      on Press: SetBit("Data_ADMIN_HMI_OKE")
      on Release: ResetBit("Data_ADMIN_HMI_OKE")
      Appearance <- "Data_ADMIN_HMI_OKE"
   Button "Button_2" at 675,175 size 122x59; TextOff '202'
      on Release: ResetBit("Data_ADMIN_HMI_Position_202")
      on Press: SetBit("Data_ADMIN_HMI_Position_202")
      Appearance <- "Data_ADMIN_HMI_CheckPosition_202"
   Button "Button_3" at 485,176 size 122x59; TextOff '201'
      on Press: SetBit("Data_ADMIN_HMI_Position_201")
      on Release: ResetBit("Data_ADMIN_HMI_Position_201")
      Appearance <- "Data_ADMIN_HMI_CheckPosition_201"
   Button "Button_4" at 674,114 size 122x59; TextOff '302'
   Button "Button_5" at 484,115 size 122x59; TextOff '301'
   Button "Button_6" at 674,54 size 122x59; TextOff '402'
   Button "Button_7" at 484,54 size 122x59; TextOff '401'
   IOField "I/O field_1" at 299,138 size 144x55; FormatPattern s99999
      ProcessValue <- "Data_ADMIN_HMI_PositionNumber"
   Button "Button_8" at 252,351 size 132x63; TextOff 'CANCEL'; TextOn 'AUTO'
      on Click: ActivateScreen("AUTO", 0)
      on Release: ResetBit("Data_ADMIN_HMI_blink_Cancel")
      on Press: SetBit("Data_ADMIN_HMI_blink_Cancel")
      Appearance <- "Data_ADMIN_HMI_blink_Cancel"
   IOField "I/O field_2" at 56,138 size 144x55; FormatPattern s99999
      ProcessValue <- "Data_Control_SlotIDFrom"
   TextField "Text field_3" at 84,204 size 74x32; Text 'FROM'
   TextField "Text field_9" at 346,204 size 57x32; Text 'TO'
   TextField "Text field_15" at 200,209 size 100x32; Text '====>'
   Button "Button_9" at 675,248 size 122x59; TextOff '102'
      on Release: ResetBit("Data_ADMIN_HMI_Position_102")
      on Press: SetBit("Data_ADMIN_HMI_Position_102")
      Appearance <- "Data_ADMIN_HMI_CheckPosition_102"
   Button "Button_10" at 485,249 size 122x59; TextOff '101'
      on Release: ResetBit("Data_ADMIN_HMI_Position_101")
      on Press: SetBit("Data_ADMIN_HMI_Position_101")
      Appearance <- "Data_ADMIN_HMI_CheckPosition_101"
*)

(* ===== HMI "HMI_RT_2" =====
system functions are stored by id; their names below are inferred from use
connection "HMI_Connection_2": S71200_TCP_IP, SCADA_S7_1200

HMI tags "Default tag table"
   "Data_Control_Elevator_SpeedManual" : Int = PLC Data_Control.Elevator.SpeedManual AT %DB5.DBW28, 500 ms
   "Data_Control_Elevator_DataSTATUSControl_INVT" : Word = PLC Data_Control.Elevator.DataSTATUSControl_INVT AT %DB5.DBW42, 500 ms
   "Data_Control_HookPallet_DataSPEEDLift_INVT" : Int = PLC Data_Control.HookPallet.DataSPEEDLift_INVT AT %DB5.DBW112, 500 ms
   "Data_Control_Elevator_DataSPEEDLift_INVT" : Int = PLC Data_Control.Elevator.DataSPEEDLift_INVT AT %DB5.DBW40, 500 ms
   "Data_Control_TableRotation_DataSpeedINVT" : Int = PLC Data_Control.TableRotation.DataSpeedINVT AT %DB5.DBW184, 500 ms
   "Data_Control_TableRotation_DataSpeedINVT_Ro" : Int = PLC Data_Control.TableRotation.DataSpeedINVT_Ro AT %DB5.DBW186, 500 ms
   "Data_Control_TableRotation_DataSpeedINVT_Down_Up" : Int = PLC Data_Control.TableRotation.DataSpeedINVT_Down_Up AT %DB5.DBW188, 500 ms
   "Data_Control_HookPallet_Hz" : Int = PLC Data_Control.HookPallet.Hz AT %DB5.DBW120, 500 ms
   "Data_Control_HookPallet_Current" : Int = PLC Data_Control.HookPallet.Current AT %DB5.DBW116, 500 ms
   "Data_Control_HookPallet_Volt" : Int = PLC Data_Control.HookPallet.Volt AT %DB5.DBW118, 500 ms
   "Data_Control_TableRotation_HZ_Ro" : Int = PLC Data_Control.TableRotation.HZ_Ro AT %DB5.DBW206, 500 ms
   "Data_Control_TableRotation_Current_Ro" : Int = PLC Data_Control.TableRotation.Current_Ro AT %DB5.DBW194, 500 ms
   "Data_Control_TableRotation_Volt_Ro" : Int = PLC Data_Control.TableRotation.Volt_Ro AT %DB5.DBW200, 500 ms
   "Data_Control_TableRotation_HZ_Up_Down" : Int = PLC Data_Control.TableRotation.HZ_Up_Down AT %DB5.DBW210, 500 ms
   "Data_Control_TableRotation_Current_Up_Down" : Int = PLC Data_Control.TableRotation.Current_Up_Down AT %DB5.DBW196, 500 ms
   "Data_Control_TableRotation_Volt_Up_Down" : Int = PLC Data_Control.TableRotation.Volt_Up_Down AT %DB5.DBW204, 500 ms
   "Data_mb_E_Data_Mb_Hz" : Int = PLC Data_mb_E.Data_Mb.Hz AT %DB29.DBW0, 500 ms
   "Data_mb_E_Data_Mb_Current" : Int = PLC Data_mb_E.Data_Mb.Current AT %DB29.DBW2, 500 ms
   "Data_mb_E_Data_Mb_Volt" : Int = PLC Data_mb_E.Data_Mb.Volt AT %DB29.DBW4, 500 ms
   "Data_MB_R_Data_Mb_Hz" : Int = PLC Data_MB_R.Data_Mb.Hz AT %DB31.DBW0, 500 ms
   "Data_MB_R_Data_Mb_Current" : Int = PLC Data_MB_R.Data_Mb.Current AT %DB31.DBW2, 500 ms
   "Data_MB_R_Data_Mb_Volt" : Int = PLC Data_MB_R.Data_Mb.Volt AT %DB31.DBW4, 500 ms
   "Data_mb_T_Data_Mb_Hz" : Int = PLC Data_mb_T.Data_Mb.Hz AT %DB30.DBW0, 500 ms
   "Data_mb_T_Data_Mb_Current" : Int = PLC Data_mb_T.Data_Mb.Current AT %DB30.DBW2, 500 ms
   "Data_mb_T_Data_Mb_Volt" : Int = PLC Data_mb_T.Data_Mb.Volt AT %DB30.DBW4, 500 ms

screen "Screen_1" 1024x768
   Button "Button_1" at 401,312 size 80x30; TextOff 'Text'

VB script "E"
   Dim objConnection
   Dim strConnectionString
   Dim GIATRI1
   Dim GIATRI2
   Dim GIATRI3
   Dim strSQL
   Dim objCommand
   
   strConnectionString = "Provider=MSDASQL;DSN=PARKINGSYSTEM;UID=sa;PWD=123456;"
    GIATRI1= HMIRuntime.SmartTags("Data_mb_E_Data_Mb_Hz")
    GIATRI2= HMIRuntime.SmartTags("Data_mb_E_Data_Mb_Current")
    GIATRI3= HMIRuntime.SmartTags("Data_mb_E_Data_Mb_Volt")
    strSQL = "UPDATE [parameter] Set valueof = " & GIATRI1 &", current_ampe = " & GIATRI2 &", voltage_v = " & GIATRI3 & " WHERE id =1"
    
   Set objConnection = CreateObject("ADODB.Connection")
   objConnection.ConnectionString = strConnectionString
   objConnection.Open
   Set objCommand = CreateObject("ADODB.Command")
   
   With objCommand
   .ActiveConnection = objConnection
   .CommandText = strSQL
   End With
   	
   objCommand.Execute
   Set objCommand = Nothing
   objConnection.Close
   Set objConnection = Nothing

VB script "Speed_T"
   Dim objConnection
   Dim strConnectionString
   Dim GIATRI1
   Dim GIATRI2
   Dim GIATRI3
   Dim strSQL
   Dim objCommand
   
   strConnectionString = "Provider=MSDASQL;DSN=PARKINGSYSTEM;UID=sa;PWD=123456;"
    GIATRI1= HMIRuntime.SmartTags("Data_mb_T_Data_Mb_Hz")
    GIATRI2= HMIRuntime.SmartTags("Data_mb_T_Data_Mb_Current")
    GIATRI3= HMIRuntime.SmartTags("Data_mb_T_Data_Mb_Volt")
    strSQL = "UPDATE [parameter] Set valueof = " & GIATRI1 &", current_ampe = " & GIATRI2 &", voltage_v = " & GIATRI3 & " WHERE id =4"
    
   Set objConnection = CreateObject("ADODB.Connection")
   objConnection.ConnectionString = strConnectionString
   objConnection.Open
   Set objCommand = CreateObject("ADODB.Command")
   
   With objCommand
   .ActiveConnection = objConnection
   .CommandText = strSQL
   End With
   	
   objCommand.Execute
   Set objCommand = Nothing
   objConnection.Close
   Set objConnection = Nothing

VB script "Speed_R"
   Dim objConnection
   Dim strConnectionString
   Dim GIATRI2
   Dim GIATRI3
   Dim GIATRI1
   Dim strSQL
   Dim objCommand
   
   strConnectionString = "Provider=MSDASQL;DSN=PARKINGSYSTEM;UID=sa;PWD=123456;"
    GIATRI1= HMIRuntime.SmartTags("Data_Control_TableRotation_HZ_Ro")
    GIATRI2= HMIRuntime.SmartTags("Data_Control_TableRotation_Current_Ro")
    GIATRI3= HMIRuntime.SmartTags("Data_Control_TableRotation_Volt_Ro")
    strSQL = "UPDATE [parameter] Set valueof = " & GIATRI1 &", current_ampe = " & GIATRI2 &", voltage_v = " & GIATRI3 & " WHERE id =3"
    
   Set objConnection = CreateObject("ADODB.Connection")
   objConnection.ConnectionString = strConnectionString
   objConnection.Open
   Set objCommand = CreateObject("ADODB.Command")
   
   With objCommand
   .ActiveConnection = objConnection
   .CommandText = strSQL
   End With
   	
   objCommand.Execute
   Set objCommand = Nothing
   objConnection.Close
   Set objConnection = Nothing

VB script "Speed_Up_Down"
   Dim objConnection
   Dim strConnectionString
   Dim GIATRI2
   Dim GIATRI1
   Dim GIATRI3
   Dim strSQL
   Dim objCommand
   
   strConnectionString = "Provider=MSDASQL;DSN=PARKINGSYSTEM;UID=sa;PWD=123456;"
    GIATRI1= HMIRuntime.SmartTags("Data_Control_TableRotation_HZ_Up_Down")
    GIATRI2= HMIRuntime.SmartTags("Data_Control_TableRotation_Current_Up_Down")
    GIATRI3= HMIRuntime.SmartTags("Data_Control_TableRotation_Volt_Up_Down")
    strSQL = "UPDATE [parameter] Set valueof = " & GIATRI1 & ", current_ampe = " & GIATRI2 &", voltage_v = " & GIATRI3 & " WHERE id =2"
    
   Set objConnection = CreateObject("ADODB.Connection")
   objConnection.ConnectionString = strConnectionString
   objConnection.Open
   Set objCommand = CreateObject("ADODB.Command")
   
   With objCommand
   .ActiveConnection = objConnection
   .CommandText = strSQL
   End With
   	
   objCommand.Execute
   Set objCommand = Nothing
   objConnection.Close
   Set objConnection = Nothing

scheduled task "Speed_E"
   on Action: "E"()
   Triggers <- "250 ms"

scheduled task "Speed_R"
   on Action: "Speed_R"()
   Triggers <- "250 ms"

scheduled task "Speed_T"
   on Action: "Speed_T"()
   Triggers <- "250 ms"

scheduled task "Speed_Up_Down"
   Triggers <- "250 ms"
   on Action: "Speed_Up_Down"()
*)